ACTION Wait_for_Part_action:
State:=STATE_RUN;
ProcessMessage01:='1IM9';(*warte auf Teil in Stopper*)
Delay.IN:=ST03_571_B69_6.BitInToCheck; 		(*  ISK an stopper.*)
Delay.PT:=T#500ms;
Delay();
END_ACTION

ACTION Wait_for_Part_exit:
ProcessMessage01:='';
END_ACTION

ACTION Close_Seperator_action:
ST03_572_Y70_0.MoveWork:=TRUE;		(* Förderband  Zuführung Vereinzler AST/GST *)
END_ACTION

ACTION Open_Stopper_action:
ST03_572_Y70_1.MoveWork:=TRUE;		(* Förderband  Züführung Stopper AST/GST *)
END_ACTION

ACTION Wait_for_Part__entry:
ProcessMessage01:='';
Delay.IN:=FALSE;
Delay();
END_ACTION

ACTION Wait_for_Part__action:
ProcessMessage01:='1IM10';(*warte auf Teil in Abholposition*)
Delay.IN:=ST03_571_B69_7.BitInToCheck; 		 (* ISK auf Abholposition Robi *)
Delay.PT:=T#500ms;
Delay();
END_ACTION

ACTION Wait_for_Part__exit:
ProcessMessage01:='';
END_ACTION

ACTION Close_Stopper_action:
ST03_572_Y70_1.MoveInit:=TRUE;		(* Förderband  Züführung Stopper AST/GST *)
END_ACTION

ACTION Open_Seperator_action:
ST03_572_Y70_0.MoveInit:=TRUE;		(* Förderband  Zuführung Vereinzler AST/GST *)
END_ACTION

ACTION SeqEnd_action:
SFCTime:=TIME_TO_DINT(TIME()-SFCTimeStart);
State:=STATE_WAIT;
END_ACTION

TRANSITION Abholpos leer:
NOT  ST03_571_B69_7.BitInToCheck		(*  ISK auf Abholposition Robi*)
END_TRANSITION

TRANSITION Part Ready:
Delay.Q AND
NOT ST03_571_B69_7.BitInToCheck	AND		(*  ISK auf Abholposition Robi*)
ST03_571_B69_6.BitInToCheck	AND				(*  ISK anwesend am Stoper*)
Robot01.ActualArea <> 4
END_TRANSITION

TRANSITION StateOk:
ST03_572_Y70_0.State=STATE_OK 	(* Förderband  Zuführung Vereinzler AST/GST *)
END_TRANSITION

TRANSITION State Ok:
ST03_572_Y70_1.State=STATE_OK 	(* Förderband  Züführung Stopper AST/GST *)
END_TRANSITION

TRANSITION Part Ready:
Delay.Q AND
Robot01.ActualArea <> 4
END_TRANSITION

TRANSITION State Ok:
ST03_572_Y70_1.State=STATE_OK 	(* Förderband  Züführung Stopper AST/GST *)
END_TRANSITION

TRANSITION StateOk:
ST03_572_Y70_0.State=STATE_OK 	(* Förderband  Zuführung Vereinzler AST/GST *)
END_TRANSITION
END_PROGRAM

(* POU zLibrary/ept/Service/_CallInit, ST *)
PROGRAM _CallInit


VAR



END_VAR
ST00_Init();
ST02_Init();
ST03_Init();

ST08_Init();
END_PROGRAM

(* POU Stations/ST_00/ST00__Init/ST00_Init, ST *)
PROGRAM ST00_Init


VAR


END_VAR
(* ----------------------------------------------------------------------------------------- *)
(* 																				Sicherungen																				 *)
(* ----------------------------------------------------------------------------------------- *)

(* Init ST00_40_F1 Vorsicherungen Leistung iO (DigIn) *)
ST00_40_F1.sInit.InstName                :='ST00_40_F1';
ST00_40_F1.sInit.Description             :='Sicherungsmodul 24VDC iO';
ST00_40_F1.sInit.BitInName               :='-40_F1';
ST00_40_F1.sInit.HomePosSignal           :=1; (* 0: Signal=Low, 1: Signal=High, 2: always  *)
ST00_40_F1.sInit.MaxTime                 :=2000;
ST00_40_F1.sInit.EnableInEveryMode       :=TRUE;

(* ----------------------------------------------------------------------------------------- *)
(* 																				Sicherheit																							 *)
(* ----------------------------------------------------------------------------------------- *)
(* Init ST03_210_S1 Not-Aus 1 Anlage ausgelöst (DigIn) *)
ST03_210_S1.sInit.InstName               :='ST03_210_S1';
ST03_210_S1.sInit.Description            :='Not-Aus 1 Anlage ausgelöst';
ST03_210_S1.sInit.BitInName              :='-210_S1';
ST03_210_S1.sInit.HomePosSignal          :=0; (* 0: Signal=Low, 1: Signal=High, 2: always  *)
ST03_210_S1.sInit.MaxTime                :=10;
ST03_210_S1.sInit.EnableInEveryMode   	 :=TRUE;

(* Init ST08_210_S2 Not-Aus 2 Anlage ausgelöst (DigIn) *)
ST08_210_S2.sInit.InstName               :='ST08_210_S2';
ST08_210_S2.sInit.Description            :='Not-Aus 2 Anlage ausgelöst';
ST08_210_S2.sInit.BitInName              :='-210_S2';
ST08_210_S2.sInit.HomePosSignal          :=1; (* 0: Signal=Low, 1: Signal=High, 2: always  *)
ST08_210_S2.sInit.MaxTime                :=10;
ST08_210_S2.sInit.EnableInEveryMode   	 :=TRUE;

(* Init ST00_X4_16 Not-Halt 2 Tampondrucker (DigIn) *)
ST00_X4_16.sInit.InstName               :='ST00_X4_16';
ST00_X4_16.sInit.Description            :='Not-Halt 2 Tampondrucker ausgelöst';
ST00_X4_16.sInit.BitInName              :='-X_16';
ST00_X4_16.sInit.HomePosSignal          :=0; (* 0: Signal=Low, 1: Signal=High, 2: always  *)
ST00_X4_16.sInit.MaxTime                :=10;
ST00_X4_16.sInit.EnableInEveryMode   	  :=TRUE;

(* Init ST00_200_A1_A1 Not-Aus iO (DigIn) *)
ST00_200_A1_A1.sInit.InstName            :='ST00_200_A1_A1';
ST00_200_A1_A1.sInit.Description         :='Not-Aus iO';
ST00_200_A1_A1.sInit.BitInName           :='-200_A1:A1';
ST00_200_A1_A1.sInit.HomePosSignal       :=1; (* 0: Signal=Low, 1: Signal=High, 2: always  *)
ST00_200_A1_A1.sInit.MaxTime             :=2000;
ST00_200_A1_A1.sInit.EnableInEveryMode   :=TRUE;

(* Init ST00_220_S1 Schutztüre 1 geöffnet (DigIn) *)
ST00_220_S1.sInit.InstName               :='ST00_220_S1';
ST00_220_S1.sInit.Description            :='Schutztüre 1 geöffnet';
ST00_220_S1.sInit.BitInName              :='-220_S1'; 
ST00_220_S1.sInit.HomePosSignal          :=0; (* 0: Signal=Low, 1: Signal=High, 2: always  *) 
ST00_220_S1.sInit.MaxTime                :=10;
ST00_220_S1.sInit.EnableInEveryMode   	 :=TRUE;

(* Init ST00_220_S2 Schutztüre 2 geöffnet (DigIn) *)
ST00_220_S2.sInit.InstName               :='ST00_220_S2';
ST00_220_S2.sInit.Description            :='Schutztüre 1 geöffnet';
ST00_220_S2.sInit.BitInName              :='-220_S2';
ST00_220_S2.sInit.HomePosSignal          :=0; (* 0: Signal=Low, 1: Signal=High, 2: always  *)
ST00_220_S2.sInit.MaxTime                :=10;
ST00_220_S2.sInit.EnableInEveryMode   	 :=TRUE;

(* Init ST00_223_S2_E1 Schutztüre 1 geschlossen (DigIn) *)
ST00_230_S2_E1.sInit.InstName            :='ST00_230_S2_E1';
ST00_230_S2_E1.sInit.Description         :='Schutztüre 1 geschlossen';
ST00_230_S2_E1.sInit.BitInName           :='-230_S2:E1';
ST00_230_S2_E1.sInit.HomePosSignal       :=2;(* :=1 @@@ *) (* 0: Signal=Low, 1: Signal=High, 2: always  *)
ST00_230_S2_E1.sInit.MaxTime             :=10;
ST00_230_S2_E1.sInit.EnableInEveryMode   	 :=TRUE;

(* Init ST00_240_S1 Schutztüre 9 geschlossen (DigIn) *)
ST00_240_S1.sInit.InstName            :='ST00_240_S1';
ST00_240_S1.sInit.Description         :='Schutztüre 9 geschlossen';
ST00_240_S1.sInit.BitInName           :='-240_S1';
ST00_240_S1.sInit.HomePosSignal       :=2;(* :=1 @@@ *) (* 0: Signal=Low, 1: Signal=High, 2: always  *)
ST00_240_S1.sInit.MaxTime             :=2000;
ST00_240_S1.sInit.EnableInEveryMode   	 :=TRUE;

(* Init ST00_226_S1 Hubtüre 1 Schleuse Einlauf STN 8 geschlossen (DigIn) *)
ST00_226_S1.sInit.InstName               :='ST00_226_S1';
ST00_226_S1.sInit.Description            :='Hubtüre 1 Schleuse Einlauf STN 8 geschlossen';
ST00_226_S1.sInit.BitInName              :='+0-226_S1';
ST00_226_S1.sInit.HomePosSignal          :=2; (* 0: Signal=Low, 1: Signal=High, 2: always  *)
ST00_226_S1.sInit.MaxTime                :=2000;
ST00_226_S1.sInit.EnableInEveryMode   	 :=TRUE;

(* Init ST00_226_S2 Hubtüre 2 Schleuse Einlauf STN 8 geschlossen (DigIn) *)
ST00_226_S2.sInit.InstName               :='ST00_226_S2';
ST00_226_S2.sInit.Description            :='Hubtüre 2 Schleuse Einlauf STN 8 geschlossen';
ST00_226_S2.sInit.BitInName              :='+0-226_S2';
ST00_226_S2.sInit.HomePosSignal          :=2; (* 0: Signal=Low, 1: Signal=High, 2: always  *)
ST00_226_S2.sInit.MaxTime                :=3000;
ST00_226_S2.sInit.EnableInEveryMode   	 :=TRUE;

(* Init ST00_227_S1 Hubtüre 3 Schleuse Auslauf STN 8 geschlossen (DigIn) *) 
ST00_227_S1.sInit.InstName               :='ST00_227_S1';
ST00_227_S1.sInit.Description            :='Hubtüre 3 Schleuse Auslauf STN 8 geschlossen';
ST00_227_S1.sInit.BitInName              :='+0-227_S1';
ST00_227_S1.sInit.HomePosSignal          :=2; (* 0: Signal=Low, 1: Signal=High, 2: always  *)
ST00_227_S1.sInit.MaxTime                :=2000;
ST00_227_S1.sInit.EnableInEveryMode   	 :=TRUE;

(* Init ST00_227_S2 Hubtüre 4 Schleuse Auslauf STN 8 geschlossen (DigIn) *)
ST00_227_S2.sInit.InstName               :='ST00_227_S2';
ST00_227_S2.sInit.Description            :='Hubtüre 4 Schleuse Auslauf STN 8 geschlossen';
ST00_227_S2.sInit.BitInName              :='+0-227_S2';
ST00_227_S2.sInit.HomePosSignal          :=2; (* 0: Signal=Low, 1: Signal=High, 2: always  *)
ST00_227_S2.sInit.MaxTime                :=2000;
ST00_227_S2.sInit.EnableInEveryMode   	 :=TRUE;

(* Init ST00_229_S1 Schutztüre Einlauf Tray STN 8 geschlossen (DigIn) *)
ST00_229_S1.sInit.InstName               :='ST00_229_S1';
ST00_229_S1.sInit.Description            :='Schutztüre Einlauf Tray STN 8 geschlossen';
ST00_229_S1.sInit.BitInName              :='+0-229_S1';
ST00_229_S1.sInit.HomePosSignal          :=2; (* 0: Signal=Low, 1: Signal=High, 2: always  *)
ST00_229_S1.sInit.MaxTime                :=2000;
ST00_229_S1.sInit.EnableInEveryMode   	 :=TRUE;

(* Init ST00_230_S1 Schutztüre Einlauf Tray STN 8 geschlossen (DigIn) *)
ST00_230_S1.sInit.InstName               :='ST00_230_S1';
ST00_230_S1.sInit.Description            :='Schutztüre Auslauf Tray STN 8 geschlossen';
ST00_230_S1.sInit.BitInName              :='+0-230_S1';
ST00_230_S1.sInit.HomePosSignal          :=2; (* 0: Signal=Low, 1: Signal=High, 2: always  *)
ST00_230_S1.sInit.MaxTime                :=2000;
ST00_230_S1.sInit.EnableInEveryMode   	 :=TRUE;

(* Init ST00_231_S1 Schutztüre Panel / Rutsche STN 8 geschlossen (DigIn) *)
ST00_231_S1.sInit.InstName               :='ST00_231_S1';
ST00_231_S1.sInit.Description            :='Schutztüre Panel / Rutsche STN 8 geschlossen';
ST00_231_S1.sInit.BitInName              :='+0-231_S1';
ST00_231_S1.sInit.HomePosSignal          :=2; (* 0: Signal=Low, 1: Signal=High, 2: always  *)
ST00_231_S1.sInit.MaxTime                :=2000;
ST00_231_S1.sInit.EnableInEveryMode   	 :=TRUE;

(* Init ST00_232_S1 Schutztüre 8 Auslauf Trays STN 8 geschlossen (DigIn) *)
ST00_232_S1.sInit.InstName               :='ST00_232_S1';
ST00_232_S1.sInit.Description            :='Schutztüre 8 Auslauf Trays STN 8 geschlossen';
ST00_232_S1.sInit.BitInName              :='+0-232_S1';
ST00_232_S1.sInit.HomePosSignal          :=2; (* 0: Signal=Low, 1: Signal=High, 2: always  *)
ST00_232_S1.sInit.MaxTime                :=2000;
ST00_232_S1.sInit.EnableInEveryMode   	 :=TRUE;

(* Init ST00_170_Motorschutz (DigIn) *)
ST00_170_Motorschutz.sInit.InstName              :='ST00_170_Motorschutz';
ST00_170_Motorschutz.sInit.Description            :='Motorschutz';
ST00_170_Motorschutz.sInit.BitInName              :='+0-170_Motorschutz';
ST00_170_Motorschutz.sInit.HomePosSignal          :=1; (* 0: Signal=Low, 1: Signal=High, 2: always  *)
ST00_170_Motorschutz.sInit.MaxTime                :=2000;
ST00_170_Motorschutz.sInit.EnableInEveryMode   	 :=TRUE;

(* Init ST00_170_Thermokontakt (DigIn) *)
ST00_170_Thermokont.sInit.InstName              :='ST00_170_Thermokont';
ST00_170_Thermokont.sInit.Description            :='Thermokontakt';
ST00_170_Thermokont.sInit.BitInName              :='+0-170_Thermokont';
ST00_170_Thermokont.sInit.HomePosSignal          :=1; (* 0: Signal=Low, 1: Signal=High, 2: always  *)
ST00_170_Thermokont.sInit.MaxTime                :=2000;
ST00_170_Thermokont.sInit.EnableInEveryMode   	 :=TRUE;

(* Init ST00_228_S1 Hubtüre 4 Schleuse Auslauf STN 8 geschlossen (DigIn) *)
ST00_228_S1.sInit.InstName               :='ST00_228_S1';
ST00_228_S1.sInit.Description            :='Pallettierer in Position';
ST00_228_S1.sInit.BitInName              :='+0-228_S1';
ST00_228_S1.sInit.HomePosSignal          :=2; (* 0: Signal=Low, 1: Signal=High, 2: always  *)
ST00_228_S1.sInit.MaxTime                :=2000;
ST00_228_S1.sInit.EnableInEveryMode   	 :=TRUE;


(* Init ST00_71_X1_3 Schnittstelle Bedrucken Tinte JSK auf Übergabeposition (DigIn) *)
ST00_71_X1_3.sInit.InstName            :='ST00_71_X1_3';
ST00_71_X1_3.sInit.Description         :='Bedrucken Tinte JSK auf Übergabeposition';
ST00_71_X1_3.sInit.BitInName           :='-71_X1_3';
ST00_71_X1_3.sInit.HomePosSignal       :=2; (* 0: Signal=Low, 1: Signal=High, 2: always  *)
ST00_71_X1_3.sInit.MaxTime             :=2000;
ST00_71_X1_3.sInit.EnableInEveryMode   :=FALSE;

(* Init ST00_71_X1_4 Schnittstelle Bedrucken Tinte Druckstation betriebsbereit (DigIn) *)
ST00_71_X1_4.sInit.InstName            :='ST00_71_X1_4';
ST00_71_X1_4.sInit.Description         :='Bedrucken Tinte Druckstation betriebsbereit';
ST00_71_X1_4.sInit.BitInName           :='-71_X1_4';
ST00_71_X1_4.sInit.HomePosSignal       :=2; (* 0: Signal=Low, 1: Signal=High, 2: always  *)
ST00_71_X1_4.sInit.MaxTime             :=2000;
ST00_71_X1_4.sInit.EnableInEveryMode   :=FALSE;

(* Init ST00_72_X1_3 Schnittstelle Tampondrucker Teil in Abholposition (DigIn) *)(*Band Entnahmeposition 1*)
ST00_72_X1_3.sInit.InstName            :='ST00_72_X1_3';
ST00_72_X1_3.sInit.Description         :='Band Entnahmeposition 1';
ST00_72_X1_3.sInit.BitInName           :='-72_X1_3';
ST00_72_X1_3.sInit.HomePosSignal       :=2; (* 0: Signal=Low, 1: Signal=High, 2: always  *)
ST00_72_X1_3.sInit.MaxTime             :=2000;
ST00_72_X1_3.sInit.EnableInEveryMode   :=FALSE;

(* Init ST00_72_X1_8 Schnittstelle Tampondrucker Druck abgeschlossen (DigIn) *)
ST00_72_X1_8.sInit.InstName            :='ST00_72_X1_8';
ST00_72_X1_8.sInit.Description         :='Tampondrucker Druck abgeschlossen';
ST00_72_X1_8.sInit.BitInName           :='-72_X1_8';
ST00_72_X1_8.sInit.HomePosSignal       :=2; (* 0: Signal=Low, 1: Signal=High, 2: always  *)
ST00_72_X1_8.sInit.MaxTime             :=2000;
ST00_72_X1_8.sInit.EnableInEveryMode   :=FALSE;

(* Init ST00_292_S1_STOP Bedienstelle Produktion Stop (DigIn) *)
ST00_292_S1_STOP.sInit.InstName          :='ST00_292_S1_STOP';
ST00_292_S1_STOP.sInit.Description       :='Bedienstelle Produktion Stop';
ST00_292_S1_STOP.sInit.BitInName         :='-292_S1:STOP';
ST00_292_S1_STOP.sInit.HomePosSignal     :=2; (* 0: Signal=Low, 1: Signal=High, 2: always  *)
ST00_292_S1_STOP.sInit.MaxTime           :=2000;
ST00_292_S1_STOP.sInit.EnableInEveryMode   	 :=TRUE;

(* Init ST00_292_S2_START Bedienstelle Produktion Start (DigIn) *)
ST00_292_S2_START.sInit.InstName         :='ST00_292_S2_START';
ST00_292_S2_START.sInit.Description      :='Bedienstelle Produktion Start';
ST00_292_S2_START.sInit.BitInName        :='-292_S2:START';
ST00_292_S2_START.sInit.HomePosSignal    :=2; (* 0: Signal=Low, 1: Signal=High, 2: always  *)
ST00_292_S2_START.sInit.MaxTime          :=2000;
ST00_292_S2_START.sInit.EnableInEveryMode   	 :=TRUE;

(* Init ST00_292_S3_RESET Bedienstelle Produktion Start (DigIn) *)
ST00_292_S3_RESET.sInit.InstName         :='ST00_292_S3_RESET';
ST00_292_S3_RESET.sInit.Description      :='Bedienstelle Produktion Reset';
ST00_292_S3_RESET.sInit.BitInName        :='-292_S3:RESET';
ST00_292_S3_RESET.sInit.HomePosSignal    :=2; (* 0: Signal=Low, 1: Signal=High, 2: always  *)
ST00_292_S3_RESET.sInit.MaxTime          :=2000;
ST00_292_S3_RESET.sInit.EnableInEveryMode   	 :=TRUE;

(* Init ST00_350_B20_0 Druckschalter Wartungseinheit Hauptluft min.6 bar (DigIn) *)
ST00_350_B20_0.sInit.InstName            :='ST00_350_B20_0';
ST00_350_B20_0.sInit.Description         :='Druckschalter Wartungseinheit Hauptluft min.6 bar';
ST00_350_B20_0.sInit.BitInName           :='-350_B20.0';
ST00_350_B20_0.sInit.HomePosSignal       :=2; (* 0: Signal=Low, 1: Signal=High, 2: always  *)
ST00_350_B20_0.sInit.MaxTime             :=2000;
ST00_350_B20_0.sInit.EnableInEveryMode   :=TRUE;

(* Init 	ST00_245_V1		Verriegelung Schutztüren-Leuchte (DigOutIn) *)
ST00_245_V1.sInit.InstName           :='ST00_245_V1';
ST00_245_V1.sInit.Description        :='Verriegelung Schutztüren';
ST00_245_V1.sInit.BitOutName         :='-245-V1';
ST00_245_V1.sInit.BitInName          :='';
ST00_245_V1.sInit.HomePosOutput      :=2; (* 0: Signal=Low, 1: Signal=High, 2: always  *)
ST00_245_V1.sInit.MaxTime            :=2000;
ST00_245_V1.sInit.EnableInEveryMode  :=TRUE;

(* Init 	ST00_245_V2_START		Bedienstelle Start-Leuchte (DigOutIn) *)
ST00_245_V2_START.sInit.InstName         :='ST00_245_V2_START';
ST00_245_V2_START.sInit.Description      :='Bedienstelle Start-Leuchte';
ST00_245_V2_START.sInit.BitOutName       :='-245_V2:START';
ST00_245_V2_START.sInit.BitInName        :='';
ST00_245_V2_START.sInit.HomePosOutput    :=2; (* 0: Signal=Low, 1: Signal=High, 2: always  *)
ST00_245_V2_START.sInit.MaxTime          :=2000;
ST00_245_V2_START.sInit.EnableInEveryMode   	 :=TRUE;

(* Init 	ST00_245_V3_RESET		Bedienstelle Reset-Schutztüren-Leuchte (DigOutIn) *)
ST00_245_V3_RESET.sInit.InstName         :='ST00_245_V3_RESET';
ST00_245_V3_RESET.sInit.Description      :='Bedienstelle Reset-Leuchte';
ST00_245_V3_RESET.sInit.BitOutName       :='-245_V3:RESET';
ST00_245_V3_RESET.sInit.BitInName        :='';
ST00_245_V3_RESET.sInit.HomePosOutput    :=2; (* 0: Signal=Low, 1: Signal=High, 2: always  *)
ST00_245_V3_RESET.sInit.MaxTime          :=2000;
ST00_245_V3_RESET.sInit.EnableInEveryMode:=TRUE;

(* Init 	ST00_245_S1_STOP 	Bedienstelle Produktion Stop (DigIn) *)
ST00_245_S1_STOP.sInit.InstName          :='ST00_245_S1_STOP';
ST00_245_S1_STOP.sInit.Description       :='Bedienstelle Produktion Stop';
ST00_245_S1_STOP.sInit.BitInName         :='-245_S1:STOP';
ST00_245_S1_STOP.sInit.HomePosSignal     :=2; (* 0: Signal=Low, 1: Signal=High, 2: always  *)
ST00_245_S1_STOP.sInit.MaxTime           :=2000;
ST00_245_S1_STOP.sInit.EnableInEveryMode :=TRUE;

(* Init 	ST00_245_S2_START	Bedienstelle Produktion Start (DigIn) *)
ST00_245_S2_START.sInit.InstName         :='ST00_245_S2_START';
ST00_245_S2_START.sInit.Description      :='Bedienstelle Produktion Start';
ST00_245_S2_START.sInit.BitInName        :='-245_S2:START';
ST00_245_S2_START.sInit.HomePosSignal    :=2; (* 0: Signal=Low, 1: Signal=High, 2: always  *)
ST00_245_S2_START.sInit.MaxTime          :=2000;
ST00_245_S2_START.sInit.EnableInEveryMode:=TRUE;

(* Init 	ST00_245_S3_RESET	Bedienstelle Produktion Reset (DigIn) *)
ST00_245_S3_RESET.sInit.InstName         :='ST00_245_S3_RESET';
ST00_245_S3_RESET.sInit.Description      :='Bedienstelle Produktion Reset';
ST00_245_S3_RESET.sInit.BitInName        :='-245_S3:RESET';
ST00_245_S3_RESET.sInit.HomePosSignal    :=2; (* 0: Signal=Low, 1: Signal=High, 2: always  *)
ST00_245_S3_RESET.sInit.MaxTime			 :=2000;
ST00_245_S3_RESET.sInit.EnableInEveryMode:=TRUE;


(* ----------------------------------------------------------------------------------------- *)
(* 																			Ausgänge																						 *)
(* ----------------------------------------------------------------------------------------- *)

(* Init ST00_31_K1 Beleuchtung Anlage (DigOutIn) *)
ST00_31_K1.sInit.InstName                :='ST00_31_K1';
ST00_31_K1.sInit.Description             :='Beleuchtung Anlage';
ST00_31_K1.sInit.BitOutName              :='-31_K1'; 
ST00_31_K1.sInit.BitInName               :='';
ST00_31_K1.sInit.HomePosOutput           :=2; (* 0: Signal=Low, 1: Signal=High, 2: always  *)
ST00_31_K1.sInit.MaxTime                 :=2000;
ST00_31_K1.sInit.EnableInEveryMode   	 	:=TRUE;
ST00_31_K1.sInit.EnableVisuInEveryMode   :=TRUE;

(* Init ST00_350_H1 Signalsäule RD Maschine Alarm/Störung (DigOutIn) *)
ST00_350_H1.sInit.InstName               :='ST00_350_H1';
ST00_350_H1.sInit.Description            :='Signalsäule RD Maschine Alarm/Störung';
ST00_350_H1.sInit.BitOutName             :='-350_H1'; 
ST00_350_H1.sInit.BitInName              :=''; 
ST00_350_H1.sInit.HomePosOutput          :=2; (* 0: Signal=Low, 1: Signal=High, 2: always  *)
ST00_350_H1.sInit.MaxTime                :=2000;
ST00_350_H1.sInit.EnableInEveryMode   	 :=TRUE;

(* Init ST00_350_H2 Signalsäule YE Bedienereingriff erforderlich (DigOutIn) *)
ST00_350_H2.sInit.InstName               :='ST00_350_H2';
ST00_350_H2.sInit.Description            :='Signalsäule YE Bedienereingriff erforderlich';
ST00_350_H2.sInit.BitOutName             :='-350_H2';
ST00_350_H2.sInit.BitInName              :='';
ST00_350_H2.sInit.HomePosOutput          :=2; (* 0: Signal=Low, 1: Signal=High, 2: always  *)
ST00_350_H2.sInit.MaxTime                :=2000;
ST00_350_H2.sInit.EnableInEveryMode   	 :=TRUE;

(* Init ST00_350_H3 Signalsäule GN Maschine Automatik (DigOutIn) *)
ST00_350_H3.sInit.InstName               :='ST00_350_H3';
ST00_350_H3.sInit.Description            :='Signalsäule GN Maschine Automatik';
ST00_350_H3.sInit.BitOutName             :='-350_H3'; 
ST00_350_H3.sInit.BitInName              :=''; 
ST00_350_H3.sInit.HomePosOutput          :=2; (* 0: Signal=Low, 1: Signal=High, 2: always  *)
ST00_350_H3.sInit.MaxTime                :=2000;
ST00_350_H3.sInit.EnableInEveryMode   	 :=TRUE;

(* Init ST00_200_A1_E4 Quittierung Not-Aus (DigOutIn) *)
ST00_200_A1_E4.sInit.InstName            :='ST00_200_A1_E4';
ST00_200_A1_E4.sInit.Description         :='Quittierung Not-Aus';
ST00_200_A1_E4.sInit.BitOutName          :='-200_A1:E4'; 
ST00_200_A1_E4.sInit.BitInName           :=''; 
ST00_200_A1_E4.sInit.HomePosSignal       :=0; (* 0: Signal=Low, 1: Signal=High, 2: always  *)
ST00_200_A1_E4.sInit.MaxTime             :=2000;
ST00_200_A1_E4.sInit.EnableInEveryMode   :=TRUE;
ST00_200_A1_E4.sInit.EnableVisuInEveryMode :=TRUE;

(* Init ST00_220_S1_S31 Verriegelung Schutztüren (DigOutIn) *)
ST00_220_S1_S31.sInit.InstName           :='ST00_220_S1_S31';
ST00_220_S1_S31.sInit.Description        :='Verriegelung Schutztüren';
ST00_220_S1_S31.sInit.BitOutName         :='-220-S1:S31';
ST00_220_S1_S31.sInit.BitInName          :='';
ST00_220_S1_S31.sInit.HomePosOutput      :=2; (* 0: Signal=Low, 1: Signal=High, 2: always  *)
ST00_220_S1_S31.sInit.MaxTime            :=2000;
ST00_220_S1_S31.sInit.EnableInEveryMode   	 :=TRUE;

(* Init ST00_292_H2_START Bedienstelle Start-Leuchte (DigOutIn) *)
ST00_292_H2_START.sInit.InstName         :='ST00_292_H2_START';
ST00_292_H2_START.sInit.Description      :='Bedienstelle Start-Leuchte';
ST00_292_H2_START.sInit.BitOutName       :='-292_H2:START';
ST00_292_H2_START.sInit.BitInName        :='';
ST00_292_H2_START.sInit.HomePosOutput    :=2; (* 0: Signal=Low, 1: Signal=High, 2: always  *)
ST00_292_H2_START.sInit.MaxTime          :=2000;
ST00_292_H2_START.sInit.EnableInEveryMode   	 :=TRUE;

(* Init ST00_292_H3_RESET Bedienstelle Reset-Leuchte (DigOutIn) *)
ST00_292_H3_RESET.sInit.InstName         :='ST00_292_H3_RESET';
ST00_292_H3_RESET.sInit.Description      :='Bedienstelle Reset-Leuchte';
ST00_292_H3_RESET.sInit.BitOutName       :='-292_H3:RESET';
ST00_292_H3_RESET.sInit.BitInName        :='';
ST00_292_H3_RESET.sInit.HomePosOutput    :=2; (* 0: Signal=Low, 1: Signal=High, 2: always  *)
ST00_292_H3_RESET.sInit.MaxTime          :=2000;
ST00_292_H3_RESET.sInit.EnableInEveryMode   	 :=TRUE;

(* Init ST00_71_K2 Schnittstelle Bedrucken Tinte Abholposition frei (DigOutIn) *)
ST00_71_K2.sInit.InstName             :='ST00_71_K2';
ST00_71_K2.sInit.Description          :='Bedrucken Tinte Abholposition frei';
ST00_71_K2.sInit.BitOutName           :='-71_K1';
ST00_71_K2.sInit.BitInName            :='';
ST00_71_K2.sInit.HomePosSignal        :=2; (* 0: Signal=Low, 1: Signal=High, 2: always  *)
ST00_71_K2.sInit.HomePosOutput	 :=2; (* 0: Signal=Low, 1: Signal=High, 2: always  *)
ST00_71_K2.sInit.MaxTime              :=2000;
ST00_71_K2.sInit.EnableVisuInEveryMode:=TRUE;

(* Schnittstelle Förderband frei für Spritzmaschine(DigOutIn) *)
ST00_73_K3.sInit.InstName             :='ST00_73_K3';
ST00_73_K3.sInit.Description          :='Förderband frei für Spritzmaschine';
ST00_73_K3.sInit.BitOutName           :='-73_K3';
ST00_73_K3.sInit.BitInName            :='';
ST00_73_K3.sInit.HomePosSignal        :=2; (* 0: Signal=Low, 1: Signal=High, 2: always  *)
ST00_73_K3.sInit.HomePosOutput				:=2; (* 0: Signal=Low, 1: Signal=High, 2: always  *)
ST00_73_K3.sInit.MaxTime              :=2000;

(*ST00_73_K4  Schnittstelle Freigabe von Spritzmaschine (nur für Anlagen ohne Rundtisch) (DigIn)*)
ST00_73_K4.sInit.InstName                :='ST00_73_K4';
ST00_73_K4.sInit.Description             :=' Freigabe Spritzmaschine';
ST00_73_K4.sInit.BitInName               :='-73_K4';
ST00_73_K4.sInit.HomePosSignal   	 :=2; (* 0: Signal=Low, 1: Signal=High, 2: always  *)
ST00_73_K4.sInit.MaxTime                 :=2000;

(* Init ST00_74_B7_2 Stopper GST1 DS (ValveSensor) *)
ST00_74_B7_2.sInit.InstName            :='ST00_74_B7_2';
ST00_74_B7_2.sInit.BitName            :='+0_74_B7_2';
ST00_74_B7_2.sInit.Description         :='Stopper GST1 DS';
ST00_74_B7_2.sInit.SensorType          :=sValveSensorType_INIT;

(* Init ST00_74_B7_3 Stopper GST1 DS (ValveSensor) *)
ST00_74_B7_3.sInit.InstName            :='ST00_74_B7_3';
ST00_74_B7_3.sInit.BitName            :='+0_74_B7_3';
ST00_74_B7_3.sInit.Description         :='Stopper GST2 PS';
ST00_74_B7_3.sInit.SensorType          :=sValveSensorType_INIT;

(* Init ST00_74_B7_4 Vereinzeler AST1 DS (ValveSensor) *)
ST00_74_B7_4.sInit.InstName            :='ST00_74_B7_4';
ST00_74_B7_4.sInit.BitName            :='+0_74_B7_4';
ST00_74_B7_4.sInit.Description         :='Vereinzeler GST1 DS';
ST00_74_B7_4.sInit.SensorType          :=sValveSensorType_INIT;

(* Init ST00_74_B7_5 Vereinzeler AST2 PS (ValveSensor) *)
ST00_74_B7_5.sInit.InstName            :='ST00_74_B7_5';
ST00_74_B7_5.sInit.BitName            :='+0_74_B7_5';
ST00_74_B7_5.sInit.Description         :='Vereinzeler GST2 PS';
ST00_74_B7_5.sInit.SensorType          :=sValveSensorType_INIT;

(* Init ST00_74_B7_6  Vereinzeler GST1 DS(ValveSensor) *)
ST00_74_B7_6.sInit.InstName            :='ST00_74_B7_6';
ST00_74_B7_6.sInit.BitName            :='+0_74_B7_6';
ST00_74_B7_6.sInit.Description         :='Vereinzeler AST1 DS';
ST00_74_B7_6.sInit.SensorType          :=sValveSensorType_WORK;

(* Init ST00_74_B7_7 Vereinzeler GST2 PS (ValveSensor) *)
ST00_74_B7_7.sInit.InstName            :='ST00_74_B7_7';
ST00_74_B7_7.sInit.BitName            :='+0_74_B7_7';
ST00_74_B7_7.sInit.Description         :='Vereinzeler AST2 PS';
ST00_74_B7_7.sInit.SensorType          :=sValveSensorType_WORK;

(* Init ST00_74_Y2_4 Stopper ISK (lt. Schaltplan 62Y1)(Valve) *)
ST00_74_Y2_4.sInit.InstName            :='ST00_74_Y2_4';
ST00_74_Y2_4.sInit.BitName            :='+0_74_Y2_4';
ST00_74_Y2_4.sInit.Description         :='Stopper Bandstrecke';
ST00_74_Y2_4.sInit.HomePosDefine       :=HOME_ALWAYS;
ST00_74_Y2_4.sInit.InitDescription     :='GS';
ST00_74_Y2_4.sInit.WorkDescription     :='AS';
ST00_74_Y2_4.sInit.DampBothTime        :=200;
ST00_74_Y2_4.sInit.KindOfValve         :='A';
ST00_74_Y2_4.sInit.MaxTime             :=2000;

(* Init ST00_74_Y2_5 Vereinzeler ISK (lt. Schaltplan 62Y3)(Valve) *)
ST00_74_Y2_5.sInit.InstName            :='ST00_74_Y2_5';
ST00_74_Y2_5.sInit.BitName            :='+0_74_Y2_5';
ST00_74_Y2_5.sInit.Description         :='Vereinzeler Bandstrecke';
ST00_74_Y2_5.sInit.HomePosDefine       :=HOME_ALWAYS;
ST00_74_Y2_5.sInit.InitDescription     :='GS';
ST00_74_Y2_5.sInit.WorkDescription     :='AS';
ST00_74_Y2_5.sInit.DampBothTime        :=200;
ST00_74_Y2_5.sInit.KindOfValve         :='A';
ST00_74_Y2_5.sInit.MaxTime             :=2000;
END_PROGRAM

(* POU Stations/ST_02_RT_Tampondrucker/ST02__Init/ST02_Init, ST *)
PROGRAM ST02_Init


VAR


END_VAR
(* ----------------------------------------------------------------------------------------- *)

(* Init ST02_S1_6A01 ST02 Sicherung 24V  (DigIn) *)
ST02_S1_6A01.sInit.InstName                :='ST02_S1_6A01';
ST02_S1_6A01.sInit.Description             :='Sicherungsmodul 24VDC';
ST02_S1_6A01.sInit.BitInName               :='-S1_6A01';
ST02_S1_6A01.sInit.HomePosSignal   :=1; (* 0: Signal=Low, 1: Signal=High, 2: always  *)
ST02_S1_6A01.sInit.MaxTime                 :=2000;
ST02_S1_6A01.sInit.EnableInEveryMode       :=TRUE;

(* ----------------------------------------------------------------------------------------- *)
(* ----------------------------------------------------------------------------------------- *)
(* Init ST02_FDB_55X1_5_READY IFM Kamera Flügelerkennung links Ready (DigIn) *)
ST02_FDB_55X1_5_READY.sInit.InstName          :='ST02_FDB_55X1_5_READY';
ST02_FDB_55X1_5_READY.sInit.Description       :='IFM Kamera links ready';
ST02_FDB_55X1_5_READY.sInit.BitInName         :='+55X1_5_READY';
ST02_FDB_55X1_5_READY.sInit.HomePosSignal     :=2; (* 0: Signal=Low, 1: Signal=High, 2: always  *)
ST02_FDB_55X1_5_READY.sInit.MaxTime           :=2000;

(* Init ST02_FDB_55X1_6_IO IFM Kamera Flügelerkennung links Ergebnis iO (DigIn) *)
ST02_FDB_55X1_6_IO.sInit.InstName          :='ST02_FDB_55X1_6_IO';
ST02_FDB_55X1_6_IO.sInit.Description       :='IFM Kamera links Ergebnis iO';
ST02_FDB_55X1_6_IO.sInit.BitInName         :='+55X1_6_IO';
ST02_FDB_55X1_6_IO.sInit.HomePosSignal     :=2; (* 0: Signal=Low, 1: Signal=High, 2: always  *)
ST02_FDB_55X1_6_IO.sInit.MaxTime           :=2000;

(* Init ST02_FDB_55X1_6_NIO IFM Kamera Flügelerkennung links Ergebnis niO (DigIn) *)
ST02_FDB_55X1_6_NIO.sInit.InstName          :='ST02_FDB_55X1_6_NIO';
ST02_FDB_55X1_6_NIO.sInit.Description       :='IFM Kamera links Ergebnis niO';
ST02_FDB_55X1_6_NIO.sInit.BitInName         :='+55X1_6_NIO';
ST02_FDB_55X1_6_NIO.sInit.HomePosSignal     :=2; (* 0: Signal=Low, 1: Signal=High, 2: always  *)
ST02_FDB_55X1_6_NIO.sInit.MaxTime           :=2000;

(* Init ST02_FDB_55X1_2_TRIGGER IFM Kamera Flügelerkennung links Trigger (DigOutIn) *)
ST02_FDB_55X1_2_TRIGGER.sInit.InstName          :='ST02_FDB_55X1_2_TRIGGER';
ST02_FDB_55X1_2_TRIGGER.sInit.Description       :='IFM Kamera links Trigger';
ST02_FDB_55X1_2_TRIGGER.sInit.BitOutName        :='+55X1_2_TRIGGER';
ST02_FDB_55X1_2_TRIGGER.sInit.BitInName         :='';
ST02_FDB_55X1_2_TRIGGER.sInit.HomePosSignal     :=2; (* 0: Signal=Low, 1: Signal=High, 2: always  *)
ST02_FDB_55X1_2_TRIGGER.sInit.MaxTime           :=2000;

(* Init ST02_FDB_55X1_7_JOB_BIT1 IFM Kamera links Jobwechsel Bit1 (DigOutIn) *)
ST02_FDB_55X1_7_JOB_BIT1.sInit.InstName          :='ST02_FDB_55X1_7_JOB_BIT1';
ST02_FDB_55X1_7_JOB_BIT1.sInit.Description       :='IFM Kamera  Job Bit 1';
ST02_FDB_55X1_7_JOB_BIT1.sInit.BitOutName        :='+55X1_7_JOB_BIT1';
ST02_FDB_55X1_7_JOB_BIT1.sInit.BitInName         :='';
ST02_FDB_55X1_7_JOB_BIT1.sInit.HomePosSignal     :=2; (* 0: Signal=Low, 1: Signal=High, 2: always  *)
ST02_FDB_55X1_7_JOB_BIT1.sInit.MaxTime           :=2000;

(* Init ST02_FDB_55X1_7_JOB_BIT2 IFM Kamera links Jobwechsel Bit2 (DigOutIn) *)
ST02_FDB_55X1_7_JOB_BIT2.sInit.InstName          :='ST02_FDB_55X1_7_JOB_BIT2';
ST02_FDB_55X1_7_JOB_BIT2.sInit.Description       :='IFM Kamera  Job Bit 2';
ST02_FDB_55X1_7_JOB_BIT2.sInit.BitOutName        :='+55X1_7_JOB_BIT2';
ST02_FDB_55X1_7_JOB_BIT2.sInit.BitInName         :='';
ST02_FDB_55X1_7_JOB_BIT2.sInit.HomePosSignal     :=2; (* 0: Signal=Low, 1: Signal=High, 2: always  *)
ST02_FDB_55X1_7_JOB_BIT2.sInit.MaxTime           :=2000;
(* Init ST02_FDB_56X1_5_READY IFM Kamera Flügelerkennung rechts Ready (DigIn) *)
ST02_FDB_56X1_5_READY.sInit.InstName          :='ST02_FDB_56X1_5_READY';
ST02_FDB_56X1_5_READY.sInit.Description       :='IFM Kamera rechts ready';
ST02_FDB_56X1_5_READY.sInit.BitInName         :='+56X1_5_READY';
ST02_FDB_56X1_5_READY.sInit.HomePosSignal     :=2; (* 0: Signal=Low, 1: Signal=High, 2: always  *)
ST02_FDB_56X1_5_READY.sInit.MaxTime           :=2000;

(* Init ST02_FDB_56X1_6_IO IFM Kamera Flügelerkennung rechts Ergebnis iO (DigIn) *)
ST02_FDB_56X1_6_IO.sInit.InstName          :='ST02_FDB_56X1_6_IO';
ST02_FDB_56X1_6_IO.sInit.Description       :='IFM Kamera rechts Ergebnis iO';
ST02_FDB_56X1_6_IO.sInit.BitInName         :='+56X1_6_IO';
ST02_FDB_56X1_6_IO.sInit.HomePosSignal     :=2; (* 0: Signal=Low, 1: Signal=High, 2: always  *)
ST02_FDB_56X1_6_IO.sInit.MaxTime           :=2000;

(* Init ST02_FDB_56X1_6_NIO IFM Kamera Flügelerkennung rechts Ergebnis niO (DigIn) *)
ST02_FDB_56X1_6_NIO.sInit.InstName          :='ST02_FDB_56X1_6_NIO';
ST02_FDB_56X1_6_NIO.sInit.Description       :='IFM Kamera rechts Ergebnis niO';
ST02_FDB_56X1_6_NIO.sInit.BitInName         :='+56X1_6_NIO';
ST02_FDB_56X1_6_NIO.sInit.HomePosSignal     :=2; (* 0: Signal=Low, 1: Signal=High, 2: always  *)
ST02_FDB_56X1_6_NIO.sInit.MaxTime           :=2000;

(* Init ST02_FDB_56X1_2_TRIGGER IFM Kamera Flügelerkennung rechts Trigger (DigOutIn) *)
ST02_FDB_56X1_2_TRIGGER.sInit.InstName          :='ST02_FDB_56X1_2_TRIGGER';
ST02_FDB_56X1_2_TRIGGER.sInit.Description       :='IFM Kamera rechts Trigger';
ST02_FDB_56X1_2_TRIGGER.sInit.BitOutName        :='+56X1_2_TRIGGER';
ST02_FDB_56X1_2_TRIGGER.sInit.BitInName         :='';
ST02_FDB_56X1_2_TRIGGER.sInit.HomePosSignal     :=2; (* 0: Signal=Low, 1: Signal=High, 2: always  *)
ST02_FDB_56X1_2_TRIGGER.sInit.MaxTime           :=2000;

(* Init ST02_FDB_56X1_7_JOB_BIT1 IFM Kamera rechts Jobwechsel Bit1 (DigOutIn) *)
ST02_FDB_56X1_7_JOB_BIT1.sInit.InstName          :='ST02_FDB_56X1_7_JOB_BIT1';
ST02_FDB_56X1_7_JOB_BIT1.sInit.Description       :='IFM Kamera  Job Bit 1';
ST02_FDB_56X1_7_JOB_BIT1.sInit.BitOutName        :='+56X1_7_JOB_BIT1';
ST02_FDB_56X1_7_JOB_BIT1.sInit.BitInName         :='';
ST02_FDB_56X1_7_JOB_BIT1.sInit.HomePosSignal     :=2; (* 0: Signal=Low, 1: Signal=High, 2: always  *)
ST02_FDB_56X1_7_JOB_BIT1.sInit.MaxTime           :=2000;

(* Init ST02_FDB_56X1_7_JOB_BIT2 IFM Kamera rechts Jobwechsel Bit2 (DigOutIn) *)
ST02_FDB_56X1_7_JOB_BIT2.sInit.InstName          :='ST02_FDB_56X1_7_JOB_BIT2';
ST02_FDB_56X1_7_JOB_BIT2.sInit.Description       :='IFM Kamera  Job Bit 2';
ST02_FDB_56X1_7_JOB_BIT2.sInit.BitOutName        :='+56X1_7_JOB_BIT2';
ST02_FDB_56X1_7_JOB_BIT2.sInit.BitInName         :='';
ST02_FDB_56X1_7_JOB_BIT2.sInit.HomePosSignal     :=2; (* 0: Signal=Low, 1: Signal=High, 2: always  *)
ST02_FDB_56X1_7_JOB_BIT2.sInit.MaxTime           :=2000;

(* Init ST02_FDB_54_B41 Kamera ISK anwesend an Prüfposition (DigIn) *)
ST02_FDB_54_B41.sInit.InstName          :='ST02_FDB_54_B41';
ST02_FDB_54_B41.sInit.Description       :='Kamera ISK an Prüfposition';
ST02_FDB_54_B41.sInit.BitInName         :='+54B41';
ST02_FDB_54_B41.sInit.HomePosSignal     :=2; (* 0: Signal=Low, 1: Signal=High, 2: always  *)
ST02_FDB_54_B41.sInit.MaxTime           :=2000;

(* Init ST02_DT_65B11 Tampondrucker Nest 1 leer (DigIn) *)
ST02_DT_65B11.sInit.InstName            :='ST02_DT_65B11';
ST02_DT_65B11.sInit.Description         :='Tampondrucker Nest 1 leer';
ST02_DT_65B11.sInit.BitInName           :='+65B11';
ST02_DT_65B11.sInit.HomePosSignal       :=2; (* 0: Signal=Low, 1: Signal=High, 2: always  *)
ST02_DT_65B11.sInit.MaxTime             :=2000;
ST02_DT_65B11.sInit.EnableInEveryMode   :=FALSE;

(* Init ST02_DT_65B21 Tampondrucker Nest 2 leer (DigIn) *)
ST02_DT_65B21.sInit.InstName            :='ST02_DT_65B21';
ST02_DT_65B21.sInit.Description         :='Tampondrucker Nest 2 leer';
ST02_DT_65B21.sInit.BitInName           :='+65B21';
ST02_DT_65B21.sInit.HomePosSignal       :=2; (* 0: Signal=Low, 1: Signal=High, 2: always  *)
ST02_DT_65B21.sInit.MaxTime             :=2000;
ST02_DT_65B21.sInit.EnableInEveryMode   :=FALSE;

(* Init ST02_S1_70K61_A1 Start Bedruckung (DigOutIn) *)
ST02_S1_70K61_A1.sInit.InstName          :='ST02_S1_70K61_A1';
ST02_S1_70K61_A1.sInit.Description       :='Start Bedruckung';
ST02_S1_70K61_A1.sInit.BitOutName        :='+70K61_A1';
ST02_S1_70K61_A1.sInit.BitInName         :='';
ST02_S1_70K61_A1.sInit.HomePosSignal     :=0; (* 0: Signal=Low, 1: Signal=High, 2: always  *)
ST02_S1_70K61_A1.sInit.MaxTime         		:=2000;

(*ST02_S1_40K01 Freigabe Förderband von SPM (DigIn)*)
ST02_S1_40K01.sInit.InstName                :='ST02_S1_40K01';
ST02_S1_40K01.sInit.Description             :=' Freigabe Förderband von SPM';
ST02_S1_40K01.sInit.BitInName               :='-S1_40K01_14';
ST02_S1_40K01.sInit.HomePosSignal    :=2; (* 0: Signal=Low, 1: Signal=High, 2: always  *)
ST02_S1_40K01.sInit.MaxTime                 :=2000;

(* Init ST02_FDB_80_B02 Band Entnahmeposition 2  (DigIn) *)
ST02_FDB_80_B02.sInit.InstName                :='ST02_FDB_80_B02';
ST02_FDB_80_B02.sInit.Description             :=' Band Entnahmeposition 2';
ST02_FDB_80_B02.sInit.BitInName               :='-80_B02';
ST02_FDB_80_B02.sInit.HomePosSignal    :=2; (* 0: Signal=Low, 1: Signal=High, 2: always  *)
ST02_FDB_80_B02.sInit.MaxTime                 :=2000;

(* Init ST02_35_S31 ST02 Druckschalter Wartungseinheit Hauptluft min.6 bar (DigIn) *)
ST02_35_S31.sInit.InstName            :='ST02_35_S31';
ST02_35_S31.sInit.Description         :='ST02 Druckschalter Wartungseinheit Hauptluft min.6 bar';
ST02_35_S31.sInit.BitInName           :='-35_S31';
ST02_35_S31.sInit.HomePosSignal       :=2; (* 0: Signal=Low, 1: Signal=High, 2: always  *)
ST02_35_S31.sInit.MaxTime             :=2000;
ST02_35_S31.sInit.EnableInEveryMode   :=TRUE;

(*---------------------------------------------------------------------------------------------------------------*)
(* Init ST02_62_Y6 Tisch drehen 0 - 180 Grad(Valve) *)
ST02_62_Y6.sInit.InstName            :='ST02_62_Y6';
ST02_62_Y6.sInit.BitName            :='+62Y6';
ST02_62_Y6.sInit.Description         :='Tisch drehen ';
ST02_62_Y6.sInit.HomePosDefine       :=HOME_ALWAYS;
ST02_62_Y6.sInit.InitDescription     :='0 Grad';
ST02_62_Y6.sInit.WorkDescription     :='180 Grad';
ST02_62_Y6.sInit.DampBothTime        :=200;
ST02_62_Y6.sInit.KindOfValve         :='2G';
ST02_62_Y6.sInit.MaxTime             :=2000;

(* Init ST02_FDB_40_B61 Iso von SPM auf Band abgelegt (DigIn) *)
ST02_FDB_40_B61.sInit.InstName            :='ST02_FDB_40_B61';
ST02_FDB_40_B61.sInit.Description         :=' Iso von SPM auf Band abgelegt';
ST02_FDB_40_B61.sInit.BitInName           :='+40B61';
ST02_FDB_40_B61.sInit.HomePosSignal       :=2; (* 0: Signal=Low, 1: Signal=High, 2: always  *)
ST02_FDB_40_B61.sInit.MaxTime             :=2000;
(*ST02_FDB_40_B61.sInit.EnableInEveryMode   :=FALSE;*)

(* Init ST02_FDB_40_B71 Iso auf Band vor Vereinzler (DigIn) *)
ST02_FDB_40_B71.sInit.InstName            :='ST02_FDB_40_B71';
ST02_FDB_40_B71.sInit.Description         :=' Iso auf Band vor Vereinzler';
ST02_FDB_40_B71.sInit.BitInName           :='+40B71';
ST02_FDB_40_B71.sInit.HomePosSignal       :=2; (* 0: Signal=Low, 1: Signal=High, 2: always  *)
ST02_FDB_40_B71.sInit.MaxTime             :=2000;
(*ST02_FDB_40_B71.sInit.EnableInEveryMode   :=FALSE;*)

(* Init ST02_DT_62_B81 Tisch drehen 0 Grad (ValveSensor) *)
ST02_DT_62_B81.sInit.InstName            :='ST02_DT_62_B81';
ST02_DT_62_B81.sInit.BitName            :='+62B81';
ST02_DT_62_B81.sInit.Description         :='Tisch drehen 0 Grad';
ST02_DT_62_B81.sInit.SensorType          :=sValveSensorType_INIT;

(* Init ST02_DT_62_B91 Tisch drehen 180 Grad (ValveSensor) *)
ST02_DT_62_B91.sInit.InstName            :='ST02_DT_62_B91';
ST02_DT_62_B91.sInit.BitName            :='+62B91';
ST02_DT_62_B91.sInit.Description         :='Tisch drehen 180 Grad';
ST02_DT_62_B91.sInit.SensorType          :=sValveSensorType_WORK;

(*---------------------------------------------------------------------------------------------------------------*)
(* Init ST02_62_Y9 Schwenkarm 2 drehen 90 - 180 Grad(Valve) *)
ST02_62_Y9.sInit.InstName            :='ST02_62_Y9';
ST02_62_Y9.sInit.BitName            :='+62Y9';
ST02_62_Y9.sInit.Description         :='Schwenkarm 2 drehen 90 - 180 Grad ';
ST02_62_Y9.sInit.HomePosDefine       :=HOME_ALWAYS;
ST02_62_Y9.sInit.InitDescription     :='90 Grad';
ST02_62_Y9.sInit.WorkDescription     :='180 Grad';
ST02_62_Y9.sInit.DampBothTime        :=200;
ST02_62_Y9.sInit.KindOfValve         :='2G';
ST02_62_Y9.sInit.MaxTime             :=2000;

(* Init ST02_62_Y11 Schwenkarm 2 drehen 90 - 0 Grad(Valve) *)
ST02_62_Y11.sInit.InstName            :='ST02_62_Y11';
ST02_62_Y11.sInit.BitName            :='+62Y11';
ST02_62_Y11.sInit.Description         :='Schwenkarm 2 drehen 90 - 0 Grad ';
ST02_62_Y11.sInit.HomePosDefine       :=HOME_ALWAYS;
ST02_62_Y11.sInit.InitDescription     :='90 Grad';
ST02_62_Y11.sInit.WorkDescription     :='0 Grad';
ST02_62_Y11.sInit.DampBothTime        :=200;
ST02_62_Y11.sInit.KindOfValve         :='2G';
ST02_62_Y11.sInit.MaxTime             :=2000;

(* Init ST02_DT_61_B31 Schwenkarm 2 0 Grad (ValveSensor) *)
ST02_DT_61_B31.sInit.InstName            :='ST02_DT_61_B31';
ST02_DT_61_B31.sInit.BitName            :='+61B31';
ST02_DT_61_B31.sInit.Description         :='Schwenkarm 2 0 Grad';
ST02_DT_61_B31.sInit.SensorType          :=sValveSensorType_WORK;

(* Init ST02_DT_61_B11 Schwenkarm 2 180 Grad (ValveSensor) *)
ST02_DT_61_B11.sInit.InstName            :='ST02_DT_61_B11';
ST02_DT_61_B11.sInit.BitName            :='+61B11';
ST02_DT_61_B11.sInit.Description         :='Schwenkarm 2 180 Grad';
ST02_DT_61_B11.sInit.SensorType          :=sValveSensorType_WORK;

(*---------------------------------------------------------------------------------------------------------------*)
(* Init ST02_62_Y13 Schwenkarm 1 drehen 90 - 180 Grad(Valve) *)
ST02_62_Y13.sInit.InstName            :='ST02_62_Y13';
ST02_62_Y13.sInit.BitName            :='+62Y13';
ST02_62_Y13.sInit.Description         :='Schwenkarm 1 drehen 90 - 180 Grad ';
ST02_62_Y13.sInit.HomePosDefine       :=HOME_ALWAYS;
ST02_62_Y13.sInit.InitDescription     :='90 Grad';
ST02_62_Y13.sInit.WorkDescription     :='180 Grad';
ST02_62_Y13.sInit.DampBothTime        :=200;
ST02_62_Y13.sInit.KindOfValve         :='2G';
ST02_62_Y13.sInit.MaxTime             :=2000;

(* Init ST02_62_Y15 Schwenkarm 1 drehen 90 - 0 Grad(Valve) *)
ST02_62_Y15.sInit.InstName            :='ST02_62_Y15';
ST02_62_Y15.sInit.BitName            :='+62Y15';
ST02_62_Y15.sInit.Description         :='Schwenkarm 1 drehen 90 - 0 Grad ';
ST02_62_Y15.sInit.HomePosDefine       :=HOME_ALWAYS;
ST02_62_Y15.sInit.InitDescription     :='90 Grad';
ST02_62_Y15.sInit.WorkDescription     :='0 Grad';
ST02_62_Y15.sInit.DampBothTime        :=200;
ST02_62_Y15.sInit.KindOfValve         :='2G';
ST02_62_Y15.sInit.MaxTime             :=2000;

(* Init ST02_DT_62_B11 Schwenkarm 1 0 Grad (ValveSensor) *)
ST02_DT_62_B11.sInit.InstName            :='ST02_DT_62_B11';
ST02_DT_62_B11.sInit.BitName            :='+62B11';
ST02_DT_62_B11.sInit.Description         :='Schwenkarm 1 0 Grad';
ST02_DT_62_B11.sInit.SensorType          :=sValveSensorType_WORK;

(* Init ST02_DT_61_B41 Schwenkarm 1 180 Grad (ValveSensor) *)
ST02_DT_61_B41.sInit.InstName            :='ST02_DT_61_B41';
ST02_DT_61_B41.sInit.BitName            :='+61B41';
ST02_DT_61_B41.sInit.Description         :='Schwenkarm 2 180 Grad';
ST02_DT_61_B41.sInit.SensorType          :=sValveSensorType_WORK;

(* Init ST02_62_Y4 Kamera Ausschleusen Bandstrecke (Valve) *)
ST02_62_Y4.sInit.InstName            :='ST02_62_Y4';
ST02_62_Y4.sInit.BitName            :='+62Y4';
ST02_62_Y4.sInit.Description         :='Kamera Ausschleusen';
ST02_62_Y4.sInit.HomePosDefine       :=HOME_ALWAYS;
ST02_62_Y4.sInit.InitDescription     :='GS';
ST02_62_Y4.sInit.WorkDescription     :='AS';
ST02_62_Y4.sInit.DampBothTime        :=200;
ST02_62_Y4.sInit.KindOfValve         :='2G';
ST02_62_Y4.sInit.MaxTime             :=4000;

(* Init ST02_FDB_54_B11 Kamera Ausschleusen Bandstrecke eingefahren (ValveSensor) *)
ST02_FDB_54_B11.sInit.InstName            :='ST02_FDB_54_B11';
ST02_FDB_54_B11.sInit.BitName            :='+54B11';
ST02_FDB_54_B11.sInit.Description         :='Kamera Ausschleusen';
ST02_FDB_54_B11.sInit.SensorType          :=sValveSensorType_INIT;

(* Init ST02_FDB_54_B21 Kamera Ausschleusen Bandstrecke ausgefahren (ValveSensor) *)
ST02_FDB_54_B21.sInit.InstName            :='ST02_FDB_54_B21';
ST02_FDB_54_B21.sInit.BitName            :='+54B21';
ST02_FDB_54_B21.sInit.Description         :='Kamera Ausschleusen';
ST02_FDB_54_B21.sInit.SensorType          :=sValveSensorType_WORK;



(*Init ST02_62_Y17 Schwenkarm 1 ISK Fixierung ein/ausfahren(Valve) *)
ST02_62_Y17.sInit.InstName            :='ST02_62_Y17';
ST02_62_Y17.sInit.BitName            :='+62_Y17';
ST02_62_Y17.sInit.Description         :='Iso 1 fiexieren';
ST02_62_Y17.sInit.HomePosDefine       :=HOME_ALWAYS;
ST02_62_Y17.sInit.InitDescription     :='GS';
ST02_62_Y17.sInit.WorkDescription     :='AS';
ST02_62_Y17.sInit.DampBothTime        :=200;
ST02_62_Y17.sInit.KindOfValve         :='2G';
ST02_62_Y17.sInit.MaxTime             :=4000;

(* Init ST02_S1_66_B11 Schwenkarm 1 ISK Fixierung GST (ValveSensor) *)
ST02_S1_66_B11.sInit.InstName            :='ST02_S1_66_B21';
ST02_S1_66_B11.sInit.BitName            :='+S1_66B11';
ST02_S1_66_B11.sInit.Description         :='Iso fixieren';
ST02_S1_66_B11.sInit.SensorType          :=sValveSensorType_INIT;

(* Init ST02_S1_66_B21 Schwenkarm 1 ISK Fixierung AST (ValveSensor) *)
ST02_S1_66_B21.sInit.InstName            :='ST02_S1_66_B21';
ST02_S1_66_B21.sInit.BitName            :='+S1_66B21';
ST02_S1_66_B21.sInit.Description         :='Iso fixieren';
ST02_S1_66_B21.sInit.SensorType          :=sValveSensorType_WORK;


(*Init ST02_62_Y18 Schwenkarm 2 ISK Fixierung ein/ausfahren(Valve) (Valve) *)
ST02_62_Y18.sInit.InstName            :='ST02_62_Y18';
ST02_62_Y18.sInit.BitName            :='+62_Y18';
ST02_62_Y18.sInit.Description         :='Iso 2 fiexieren';
ST02_62_Y18.sInit.HomePosDefine       :=HOME_ALWAYS;
ST02_62_Y18.sInit.InitDescription     :='GS';
ST02_62_Y18.sInit.WorkDescription     :='AS';
ST02_62_Y18.sInit.DampBothTime        :=200;
ST02_62_Y18.sInit.KindOfValve         :='2G';
ST02_62_Y18.sInit.MaxTime             :=4000;

(* Init ST02_S1_66_B31 Schwenkarm 2 ISK Fixierung GST (ValveSensor) *)
ST02_S1_66_B31.sInit.InstName            :='ST02_S1_66_B31';
ST02_S1_66_B31.sInit.BitName            :='S1_66B31';
ST02_S1_66_B31.sInit.Description         :='Iso fixieren';
ST02_S1_66_B31.sInit.SensorType          :=sValveSensorType_INIT;

(* Init ST02_S1_66_B41 Schwenkarm 2 ISK Fixierung AST (ValveSensor) *)
ST02_S1_66_B41.sInit.InstName            :='ST02_S1_66_B41';
ST02_S1_66_B41.sInit.BitName            :='S1_66_B41';
ST02_S1_66_B41.sInit.Description         :='Iso fixieren';
ST02_S1_66_B41.sInit.SensorType          :=sValveSensorType_WORK;


(* Init ST02_35Y01 Einschaltventil Hauptluft Tampondruckanlage (Valve) *)
ST02_35Y01.sInit.InstName          :='ST02_35Y01';
ST02_35Y01.sInit.BitName          :='+35Y01';
ST02_35Y01.sInit.Description       :='Hauptluft Tampondrucker';
ST02_35Y01.sInit.HomePosDefine     :=HOME_ALWAYS;
ST02_35Y01.sInit.InitDescription   :='GS';
ST02_35Y01.sInit.WorkDescription   :='AS';
ST02_35Y01.sInit.DampBothTime      :=0;
ST02_35Y01.sInit.MaxTime           :=2000;
ST02_35Y01.sInit.KindOfValve       :='A';
END_PROGRAM

(* POU Stations/ST_03_Ruestsaetze/ST_03__Init/ST03_Init, ST *)
PROGRAM ST03_Init


VAR


	sDigInVisu: BOOL;
END_VAR
(*INIT Aufrufe für Rüstsätze*)
Init_154polRP();	Init_154pol();
Init_160pol();		Init_206pol();
Init_92pol();		Init_124pol();
Init_46pol();		Init_NOX5_6pol();
Init_NOX4pol();	Init_88pol();
Init_7pol();		Init_88polAMG();
Init_120pol();		Init_21pol();
Init_191pol();		Init_48pol();
Init_72pol();		Init_268pol_102pol_neu();
Init_268polRP();	Init_33pol();

(* ----------------------------------------------------------------------------------------- *)
IF NOT MP.ST03.SGM_3621 THEN
	(*Init ST03_51_M1 Förderbandmotor*)
	ST03_51_M1.sConfig.Description		:='Förderband';
	ST03_51_M1.sConfig.InstName			:='ST03_51_M1';
	ST03_51_M1.sConfig.Aktiv				:=TRUE;
	ST03_51_M1.sConfig.Skalierfaktor		:=360.0 / (EXPT(2,20))	; (*360°/ 20 bit Encoder =0.00034332275390625*)
	ST03_51_M1.sConfig.Getriebefaktor		:=25;
	ST03_51_M1.sConfig.Modulo			:=FALSE;
	ST03_51_M1.sConfig.Pos_Faktor		:=157.07;			(*Weg bei einer Umdrehung in mm (nach Getriebe)*)
	ST03_51_M1.sConfig.maxRpm			:=5338;
	ST03_51_M1.sConfig.ModeOfOperation	:=CSP;				(*CSP,CSV,CST,CSTCA muss an der KLemme (Coe-Online 7010.03) eingestellt werden*)
	(*(CSP) position mode*)
	ST03_51_M1.sConfig.Torque_Limit		:=0;			(*bei 0 ausgeschaltet*)
	ST03_51_M1.sConfig.SW_Limit_on		:=FALSE;
	ST03_51_M1.sConfig.SW_Limit_min		:=-EXPT(2,32);
	ST03_51_M1.sConfig.SW_Limit_max		:=EXPT(2,32);
	ST03_51_M1.sConfig.lr_kp 				:= 800;
	ST03_51_M1.sConfig.lr_ki 				:= 100.0;
	ST03_51_M1.sConfig.lr_kd 				:= 50;
ELSE
	(* Init ST03_A5 Bandantrieb Förderbandmotor Oriental (nur 3621) Ein (DigOutIn)   ST08_170_K2 *)
	ST03_A5.sInit.InstName               :='ST03_A5';
	ST03_A5.sInit.Description            :='Förderbandmotor Isokörper';
	ST03_A5.sInit.BitOutName             :='-3_A5';
	ST03_A5.sInit.BitInName              :='';
	ST03_A5.sInit.HomePosOutput          :=2; (* 0: Signal=Low, 1: Signal=High, 2: always  *)
	ST03_A5.sInit.MaxTime                :=2000;
	ST03_A5.sInit.EnableInEveryMode  :=TRUE;
END_IF

(* Init ST03_V2 Störung Motor Förderband Oriental (DigIn) *)
ST03_V2.sInit.InstName               :='ST03_V2';
ST03_V2.sInit.Description            :='Störung Motor Förderband';
ST03_V2.sInit.BitInName              :='+3-V2';
ST03_V2.sInit.HomePosSignal          :=2; (* 0: Signal=Low, 1: Signal=High, 2: always  *)
ST03_V2.sInit.MaxTime                :=10;
ST03_V2.sInit.EnableInEveryMode       :=TRUE;

(* Init ST03_601V1_A1  Förderband Prüfteile (DigOutIn)  *)
ST03_601V1_A1.sInit.InstName               :='ST03_601V1_A1';
ST03_601V1_A1.sInit.Description            :='Förderband Prüfteile';
ST03_601V1_A1.sInit.BitOutName             :='-60V1_A1';
ST03_601V1_A1.sInit.BitInName              :='';
ST03_601V1_A1.sInit.HomePosOutput          :=2; (* 0: Signal=Low, 1: Signal=High, 2: always  *)
ST03_601V1_A1.sInit.MaxTime                :=2000;
ST03_601V1_A1.sInit.EnableInEveryMode  			:=TRUE;

(* ----------------------------------------------------------------------------------------- *)
(* 																	Roboter																									 *)
(* ----------------------------------------------------------------------------------------- *)
Visu.Robot01.TcpIpAdress:=MP.ST03.RobotIPAdress;
Robot01.sInit.InstName				:='Robot01';
Robot01.sInit.BitName				:='+3-125_A1';
Robot01.sInit.Description				:='ST03 Roboter';
Robot01.sInit.TcpIPAdress			:=MP.ST03.RobotIPAdress; (*10.16.55.130*)
Robot01.sInit.TcpIPSocket			:=2000;
Robot01.sInit.MaxTime				:=40000;
Robot01.sInit.WithToolHandling		:=TRUE;
Robot01.sInit.ToolMaxTime			:=2000;

(* Init ST03_125_F1 Absicherung Roboter iO (DigIn) *)
ST03_125_F1.sInit.InstName               :='ST03_125_F1';
ST03_125_F1.sInit.Description            :='Absicherung Roboter iO';
ST03_125_F1.sInit.BitInName              :='+3-125_F1';
ST03_125_F1.sInit.HomePosSignal          :=2; (* 0: Signal=Low, 1: Signal=High, 2: always  *)
ST03_125_F1.sInit.MaxTime                :=10;
ST03_125_F1.sInit.EnableInEveryMode       :=TRUE;

(* Init ST03_400_B12_6 Schwenkmodul GST (Roboterkopf) (DigIn) *)
ST03_400_B12_6.sInit.InstName           :='ST03_400_B12_6';
ST03_400_B12_6.sInit.Description        :='Rob. ST03 Schwenken GST';
ST03_400_B12_6.sInit.BitInName          :='+3-400_B12_6';
ST03_400_B12_6.sInit.HomePosSignal      :=2; (* 0: Signal=Low, 1: Signal=High, 2: always  *)
ST03_400_B12_6.sInit.MaxTime            :=2000;

(* Init ST03_400_B12_7 Schwenkmodul AST (Roboter) (DigIn) *)
ST03_400_B12_7.sInit.InstName           :='ST03_400_B12_7';
ST03_400_B12_7.sInit.Description        :='Rob. ST03 Schwenken AST';
ST03_400_B12_7.sInit.BitInName          :='+3-400_B12_7';
ST03_400_B12_7.sInit.HomePosSignal      :=2; (* 0: Signal=Low, 1: Signal=High, 2: always  *)
ST03_400_B12_7.sInit.MaxTime            :=2000;

(* Init St03_120_A1_A14 Rob. opt. Tool 2 ist Ein (DigIn) *)
St03_120_A1_A14.sInit.InstName           :='St03_120_A1_A14';
St03_120_A1_A14.sInit.Description        :='Rob. opt. Tool 2 ist Ein';
St03_120_A1_A14.sInit.BitInName          :='+3-120_A1_A14';
St03_120_A1_A14.sInit.HomePosSignal      :=2; (* 0: Signal=Low, 1: Signal=High, 2: always  *)
St03_120_A1_A14.sInit.MaxTime            :=2000;

(* Init ST03_BG3_S53_0 Start Band für Dummyprüfung (DigIn) *)
ST03_BG3_S53_0.sInit.InstName               :='ST03_BG3_S53_0';
ST03_BG3_S53_0.sInit.Description            :='Start Band für Dummyprüfung';
ST03_BG3_S53_0.sInit.BitInName              :='+0-BG3_S53_0';
ST03_BG3_S53_0.sInit.HomePosSignal          :=2; (* 0: Signal=Low, 1: Signal=High, 2: always  *)
ST03_BG3_S53_0.sInit.MaxTime                :=2000;
ST03_BG3_S53_0.sInit.EnableInEveryMode   	 :=TRUE;

(* Init ST03_BG3_X53_0 LED TasterStart Band für Dummyprüfung (DigOutIn) *)
ST03_BG3_X53_0.sInit.InstName          :='ST03_BG3_X53_0';
ST03_BG3_X53_0.sInit.Description       :='LED TasterStart Band für Dummyprüfung';
ST03_BG3_X53_0.sInit.BitOutName        :='+ST03_BG3_X53_0';
ST03_BG3_X53_0.sInit.BitInName         :='';
ST03_BG3_X53_0.sInit.HomePosSignal     :=2; (* 0: Signal=Low, 1: Signal=High, 2: always  *)
ST03_BG3_X53_0.sInit.MaxTime           :=2000;

(* Init ST03_400_B54_7 Tray Testteile in Position (DigIn) *)
ST03_400_B54_7.sInit.InstName            :='ST03_400_B54_7';
ST03_400_B54_7.sInit.Description         :='Tray Testteile in Position';
ST03_400_B54_7.sInit.BitInName           :='+8-400_B54.7';
ST03_400_B54_7.sInit.HomePosSignal       :=2; (* 0: Signal=Low, 1: Signal=High, 2: always  *)
ST03_400_B54_7.sInit.MaxTime             :=2000;

(* Init ST03_8_75_B13_5 voll/belegt keine Prüfteile mehr (DigIn) *)
ST03_8_75_B13_5.sInit.InstName            :='ST03_8_75_B13_5';
ST03_8_75_B13_5.sInit.Description         :='voll/belegt keine Prüfteile mehr';
ST03_8_75_B13_5.sInit.BitInName           :='+8-75_B13.5';
ST03_8_75_B13_5.sInit.HomePosSignal       :=2; (* 0: Signal=Low, 1: Signal=High, 2: always  *)
ST03_8_75_B13_5.sInit.MaxTime             :=2000;

(* Init ST03_8_75_B13_6 belegt mit 6 Prüfteile (DigIn) *)
ST03_8_75_B13_6.sInit.InstName            :='ST03_8_75_B13_6';
ST03_8_75_B13_6.sInit.Description         :='belegt mit 6 Prüfteile';
ST03_8_75_B13_6.sInit.BitInName           :='+8-75_B13.6';
ST03_8_75_B13_6.sInit.HomePosSignal       :=2; (* 0: Signal=Low, 1: Signal=High, 2: always  *)
ST03_8_75_B13_6.sInit.MaxTime             :=2000;

(* Init ST03_65_Q1 LED TasterStart Band für Dummyprüfung (DigOutIn) *)
ST03_65_Q1.sInit.InstName          :='ST03_65_Q1';
ST03_65_Q1.sInit.Description       :='Kühltunnel (Lüfter)';
ST03_65_Q1.sInit.BitOutName        :='+ST03_65_Q1';
ST03_65_Q1.sInit.BitInName         :='';
ST03_65_Q1.sInit.HomePosSignal     :=2; (* 0: Signal=Low, 1: Signal=High, 2: always  *)
ST03_65_Q1.sInit.MaxTime           :=2000;

(* Init ST03_65_F1 Tray Testteile in Position (DigIn) *)
ST03_65_F1.sInit.InstName            :='ST03_65_F1';
ST03_65_F1.sInit.Description         :='Sicherung Kühltunnel (Lüfter)';
ST03_65_F1.sInit.BitInName           :='+8-65_F1';
ST03_65_F1.sInit.HomePosSignal       :=2; (* 0: Signal=Low, 1: Signal=High, 2: always  *)
ST03_65_F1.sInit.MaxTime             :=2000;
END_PROGRAM
ACTION Init_120pol:
(*Rüstsatz 120 pol ==================================================================================*)

(* Init ST03_531_B69_0 Zuführung  frei zum Ablegen ISK SP Maschine (DigIn) *)
ST03_531_B69_0.sInit.InstName            :='ST03_531_B69_0';
ST03_531_B69_0.sInit.Description         :='frei zum Ablegen ISK SP Maschine';
ST03_531_B69_0.sInit.BitInName           :='+8-531_B69.0';
ST03_531_B69_0.sInit.HomePosSignal       :=2; (* 0: Signal=Low, 1: Signal=High, 2: always  *)
ST03_531_B69_0.sInit.MaxTime             :=2000;
ST03_531_B69_0.sInit.EnableInEveryMode   :=TRUE;

(* Init ST03_531_B69_1 Zuführung Vereinzler eingefahren GST (ValveSensor) *)
ST03_531_B69_1.sInit.InstName		:='ST03_531_B69_1';
ST03_531_B69_1.sInit.BitName		:='+8_531_B69.1';
ST03_531_B69_1.sInit.Description	:=' Vereinzler eingefahren GST';
ST03_531_B69_1.sInit.SensorType	:=sValveSensorType_INIT;

(* Init ST03_531_B69_2 Zuführung Vereinzler ausgefahren AST (ValveSensor) *)
ST03_531_B69_2.sInit.InstName		:='ST03_531_B69_2';
ST03_531_B69_2.sInit.BitName		:='+8_531_B69.2';
ST03_531_B69_2.sInit.Description	:=' Vereinzler ausgefahren AST';
ST03_531_B69_2.sInit.SensorType	:=sValveSensorType_WORK;

(* Init ST03_531_B69_3 Zuführung Stopper eingefahren AST (ValveSensor) *)
ST03_531_B69_3.sInit.InstName		:='ST03_531_B69_3';
ST03_531_B69_3.sInit.BitName		:='+8_531_B69.3';
ST03_531_B69_3.sInit.Description	:='Stopper eingefahren AST';
ST03_531_B69_3.sInit.SensorType	:=sValveSensorType_WORK;

(* Init ST03_531_B69_4 Zuführung Stopper ausgefahren GST (ValveSensor) *)
ST03_531_B69_4.sInit.InstName		:='ST03_531_B69_4';
ST03_531_B69_4.sInit.BitName		:='+8_531_B69.4';
ST03_531_B69_4.sInit.Description	:='Stopper ausgefahren GST';
ST03_531_B69_4.sInit.SensorType	:=sValveSensorType_INIT;;

(* Init ST03_531_B69_6 ISK anwesend am Stopper (DigIn) *)
ST03_531_B69_6.sInit.InstName            :='ST03_531_B69_6';
ST03_531_B69_6.sInit.Description         :='ISK anwesend am Stopper';
ST03_531_B69_6.sInit.BitInName           :='+8-531_B69.6';
ST03_531_B69_6.sInit.HomePosSignal       :=2; (* 0: Signal=Low, 1: Signal=High, 2: always  *)
ST03_531_B69_6.sInit.MaxTime             :=2000;
ST03_531_B69_6.sInit.EnableInEveryMode   :=TRUE;

(* Init ST03_531_B69_7 ISK rechts Lageerkennung (DigIn) *)
ST03_531_B69_7.sInit.InstName            :='ST03_531_B69_7';
ST03_531_B69_7.sInit.Description         :='ISK Lageerkennung rechts.';
ST03_531_B69_7.sInit.BitInName           :='+8-531_B69.7';
ST03_531_B69_7.sInit.HomePosSignal       :=2; (* 0: Signal=Low, 1: Signal=High, 2: always  *)
ST03_531_B69_7.sInit.MaxTime             :=2000;
ST03_531_B69_7.sInit.EnableInEveryMode   :=TRUE;

(* Init ST03_562_B70_0 ISK links Lageerkennung (DigIn) *)
ST03_532_B70_0.sInit.InstName            :='ST03_532_B70_0';
ST03_532_B70_0.sInit.Description         :='ISK Lageerkennung links';
ST03_532_B70_0.sInit.BitInName           :='+8-532_B70.0';
ST03_532_B70_0.sInit.HomePosSignal       :=2; (* 0: Signal=Low, 1: Signal=High, 2: always  *)
ST03_532_B70_0.sInit.MaxTime             :=2000;
ST03_532_B70_0.sInit.EnableInEveryMode   :=TRUE;

(* Init ST03_532_Y70_1   Zuführung  Vereinzler AST/GST (Valve) *)
ST03_532_Y70_1.sInit.InstName            :='ST03_532_Y70_1';
ST03_532_Y70_1.sInit.BitName            :='+8-532_Y70.1';
ST03_532_Y70_1.sInit.Description         :=' Zuführung Vereinzler AST/GST';
ST03_532_Y70_1.sInit.HomePosDefine       :=HOME_ALWAYS;
ST03_532_Y70_1.sInit.InitDescription     :='GS einfahren';
ST03_532_Y70_1.sInit.WorkDescription     :='AS ausfahren';
ST03_532_Y70_1.sInit.DampBothTime        :=200;
ST03_532_Y70_1.sInit.KindOfValve         :='A';
ST03_532_Y70_1.sInit.MaxTime             :=2000;

(* Init ST03_532_Y70_2   Zuführung  Stopper AST/GST (Valve) *)
ST03_532_Y70_2.sInit.InstName            :='ST03_532_Y70_2';
ST03_532_Y70_2.sInit.BitName            :='+8-532_Y70.2';
ST03_532_Y70_2.sInit.Description         :=' Zuführung Stopper AST/GST';
ST03_532_Y70_2.sInit.HomePosDefine       :=HOME_ALWAYS;
ST03_532_Y70_2.sInit.InitDescription     :='GS ausfahren';
ST03_532_Y70_2.sInit.WorkDescription     :='AS einfahren';
ST03_532_Y70_2.sInit.DampBothTime        :=200;
ST03_532_Y70_2.sInit.KindOfValve         :='A';
ST03_532_Y70_2.sInit.MaxTime             :=2000;
END_ACTION
ACTION Init_124pol:
(*========================= Rüstsatz 124 polig===============================*)

(* Init ST03_451_B69_0 Förderbandeinheit  Zuführung Vereinzler AST (ValveSensor) *)
ST03_451_B69_0.sInit.InstName            :='ST03_451_B69_0';
ST03_451_B69_0.sInit.BitName            :='+8_451_B69.0';
ST03_451_B69_0.sInit.Description         :='Förderbandeinheit  Zuführung Vereinzler AST';
ST03_451_B69_0.sInit.SensorType          :=sValveSensorType_INIT;

(* Init ST03_451_B69_1 Förderbandeinheit  Zuführung Vereinzler GST (ValveSensor) *)
ST03_451_B69_1.sInit.InstName            :='ST03_451_B69_1';
ST03_451_B69_1.sInit.BitName            :='+8_451_B69.1';
ST03_451_B69_1.sInit.Description         :='Förderbandeinheit  Zuführung Vereinzler GST';
ST03_451_B69_1.sInit.SensorType          :=sValveSensorType_WORK;

(* Init ST03_451_B69_2 Förderbandeinheit  Zuführung Stopper AST (ValveSensor) *)
ST03_451_B69_2.sInit.InstName            :='ST03_451_B69_2';
ST03_451_B69_2.sInit.BitName            :='+8_451_B69.2';
ST03_451_B69_2.sInit.Description         :='Förderband linke Zuführung Stopper AST';
ST03_451_B69_2.sInit.SensorType          :=sValveSensorType_INIT;

(* Init ST03_451_B69_3 Förderbandeinheit  Zuführung Stopper GST (ValveSensor) *)
ST03_451_B69_3.sInit.InstName            :='ST03_451_B69_3';
ST03_451_B69_3.sInit.BitName            :='+8_451_B69.3';
ST03_451_B69_3.sInit.Description         :='Förderband linke Zuführung Stopper GST';
ST03_451_B69_3.sInit.SensorType          :=sValveSensorType_WORK;

(* Init ST03_451_B69_4  Zuführung  frei zum Ablegen ISK SP Maschine Pos.1 (DigIn) *)
ST03_451_B69_4.sInit.InstName            :='ST03_451_B69_4';
ST03_451_B69_4.sInit.Description         :='Zuführung links frei zum Ablegen ISK SP Maschine Pos1';
ST03_451_B69_4.sInit.BitInName           :='+8-451_B69.4';
ST03_451_B69_4.sInit.HomePosSignal       :=2; (* 0: Signal=Low, 1: Signal=High, 2: always  *)
ST03_451_B69_4.sInit.MaxTime             :=2000;
ST03_451_B69_4.sInit.EnableInEveryMode   :=TRUE;

(* Init ST03_451_B69_7  ISK anwesend am Vereinzler (DigIn) *)
ST03_451_B69_7.sInit.InstName            :='ST03_451_B69_7';
ST03_451_B69_7.sInit.Description         :='ISK anwesend am Vereinzler';
ST03_451_B69_7.sInit.BitInName           :='+8-451_B69.7';
ST03_451_B69_7.sInit.HomePosSignal       :=2; (* 0: Signal=Low, 1: Signal=High, 2: always  *)
ST03_451_B69_7.sInit.MaxTime             :=2000;
ST03_451_B69_7.sInit.EnableInEveryMode   :=TRUE;

(* Init ST03_452_B70_1  Züführung  ISK Lageerkennung 1 (DigIn) *)
ST03_452_B70_1.sInit.InstName            :='ST03_452_B70_1';
ST03_452_B70_1.sInit.Description         :='Züführung  ISK Lageerkennung 1';
ST03_452_B70_1.sInit.BitInName           :='+8-452_B70.1';
ST03_452_B70_1.sInit.HomePosSignal       :=2; (* 0: Signal=Low, 1: Signal=High, 2: always  *)
ST03_452_B70_1.sInit.MaxTime             :=2000;
ST03_452_B70_1.sInit.EnableInEveryMode   :=TRUE;

(* Init ST03_452_B70_2  Züführung  ISK Lageerkennung 2 (DigIn) *)
ST03_452_B70_2.sInit.InstName            :='ST03_452_B70_2';
ST03_452_B70_2.sInit.Description         :='Züführung  ISK Lageerkennung 2';
ST03_452_B70_2.sInit.BitInName           :='+8-452_B70.2';
ST03_452_B70_2.sInit.HomePosSignal       :=2; (* 0: Signal=Low, 1: Signal=High, 2: always  *)
ST03_452_B70_2.sInit.MaxTime             :=2000;
ST03_452_B70_2.sInit.EnableInEveryMode   :=TRUE;

(* Init ST03_453_B70_4  ISK anwesend Übergabeposition Roboter (DigIn) *)
ST03_453_B70_4.sInit.InstName            :='ST03_453_B70_4';
ST03_453_B70_4.sInit.Description         :='Zuführung ISK auf Übergabeposition Robo Palettierer ';
ST03_453_B70_4.sInit.BitInName           :='+8-453_B70.4';
ST03_453_B70_4.sInit.HomePosSignal       :=2; (* 0: Signal=Low, 1: Signal=High, 2: always  *)
ST03_453_B70_4.sInit.MaxTime             :=2000;
ST03_453_B70_4.sInit.EnableInEveryMode   :=TRUE;

(* Init ST03_453_Y70_5 Förderband  Zuführung Vereinzler (Valve) *)
ST03_453_Y70_5.sInit.InstName            :='ST03_453_Y70_5';
ST03_453_Y70_5.sInit.BitName            :='+8-453_Y70.5';
ST03_453_Y70_5.sInit.Description         :='Förderband  Zuführung Vereinzler';
ST03_453_Y70_5.sInit.HomePosDefine       :=HOME_ALWAYS;
ST03_453_Y70_5.sInit.InitDescription     :='GS einfahren';
ST03_453_Y70_5.sInit.WorkDescription     :='AS ausfahren';
ST03_453_Y70_5.sInit.DampBothTime        :=200;
ST03_453_Y70_5.sInit.KindOfValve         :='A';
ST03_453_Y70_5.sInit.MaxTime             :=2000;

(* Init ST03_453_Y70_6 Förderband  Zuführung Stopper (Valve) *)
ST03_453_Y70_6.sInit.InstName            :='ST03_453_Y70_6';
ST03_453_Y70_6.sInit.BitName            :='+8-453_Y70.6';
ST03_453_Y70_6.sInit.Description         :='Förderband  Zuführung Stopper';
ST03_453_Y70_6.sInit.HomePosDefine       :=HOME_ALWAYS;
ST03_453_Y70_6.sInit.InitDescription     :='GS ausfahren';
ST03_453_Y70_6.sInit.WorkDescription     :='AS einfahren';
ST03_453_Y70_6.sInit.DampBothTime        :=200;
ST03_453_Y70_6.sInit.KindOfValve         :='A';
ST03_453_Y70_6.sInit.MaxTime             :=2000;
END_ACTION
ACTION Init_154pol:
(*Rüstsatz 154pol*)
(* Init ST03_425_B67_0 Förderbandeinheit  Zuführung Vereinzler AST (ValveSensor) *)
ST03_425_B67_0.sInit.InstName            :='ST03_425_B67_0';
ST03_425_B67_0.sInit.BitName            :='+8_425_B67.0';
ST03_425_B67_0.sInit.Description         :='Förderbandeinheit  Zuführung Vereinzler AST';
ST03_425_B67_0.sInit.SensorType          :=sValveSensorType_INIT;

(* Init ST03_425_B67_1 Förderbandeinheit  Zuführung Vereinzler GST (ValveSensor) *)
ST03_425_B67_1.sInit.InstName            :='ST03_425_B67_1';
ST03_425_B67_1.sInit.BitName            :='+8_425_B67.1';
ST03_425_B67_1.sInit.Description         :='Förderbandeinheit  Zuführung Vereinzler GST';
ST03_425_B67_1.sInit.SensorType          :=sValveSensorType_WORK;

(* Init ST03_425_B67_2 Förderbandeinheit  Zuführung Stopper AST (ValveSensor) *)
ST03_425_B67_2.sInit.InstName            :='ST03_425_B67_2';
ST03_425_B67_2.sInit.BitName            :='+8_425_B67.2';
ST03_425_B67_2.sInit.Description         :='Förderband linke Zuführung Stopper AST';
ST03_425_B67_2.sInit.SensorType          :=sValveSensorType_INIT;

(* Init ST03_425_B67_3 Förderbandeinheit  Zuführung Stopper GST (ValveSensor) *)
ST03_425_B67_3.sInit.InstName            :='ST03_425_B67_3';
ST03_425_B67_3.sInit.BitName            :='+8_425_B67.3';
ST03_425_B67_3.sInit.Description         :='Förderband linke Zuführung Stopper GST';
ST03_425_B67_3.sInit.SensorType          :=sValveSensorType_WORK;

(* Init ST03_425_B67_4  Zuführung  frei zum Ablegen ISK SP Maschine Pos.1 (DigIn) *)
ST03_425_B67_4.sInit.InstName            :='ST03_425_B67_4';
ST03_425_B67_4.sInit.Description         :='Zuführung links frei zum Ablegen ISK SP Maschine Pos1';
ST03_425_B67_4.sInit.BitInName           :='+8-425_B67.4';
ST03_425_B67_4.sInit.HomePosSignal       :=2; (* 0: Signal=Low, 1: Signal=High, 2: always  *)
ST03_425_B67_4.sInit.MaxTime             :=2000;
ST03_425_B67_4.sInit.EnableInEveryMode   :=TRUE;

(* Init ST03_425_B67_5  Zuführung  frei zum Ablegen ISK SP Maschine Pos.2 (DigIn) *)
ST03_425_B67_5.sInit.InstName            :='ST03_425_B67_5';
ST03_425_B67_5.sInit.Description         :='Zuführung links frei zum Ablegen ISK SP Maschine Pos2';
ST03_425_B67_5.sInit.BitInName           :='+8-425_B67.5';
ST03_425_B67_5.sInit.HomePosSignal       :=2; (* 0: Signal=Low, 1: Signal=High, 2: always  *)
ST03_425_B67_5.sInit.MaxTime             :=2000;
ST03_425_B67_5.sInit.EnableInEveryMode   :=TRUE;

(* Init ST03_425_B67_6  Zuführung  frei zum Ablegen ISK SP Maschine Pos.3 (DigIn) *)
ST03_425_B67_6.sInit.InstName            :='ST03_425_B67_6';
ST03_425_B67_6.sInit.Description         :='Zuführung links frei zum Ablegen ISK SP Maschine Pos3';
ST03_425_B67_6.sInit.BitInName           :='+8-425_B67.6';
ST03_425_B67_6.sInit.HomePosSignal       :=2; (* 0: Signal=Low, 1: Signal=High, 2: always  *)
ST03_425_B67_6.sInit.MaxTime             :=2000;
ST03_425_B67_6.sInit.EnableInEveryMode   :=TRUE;

(* Init ST03_425_B67_7  ISK anwesend am Vereinzler (DigIn) *)
ST03_425_B67_7.sInit.InstName            :='ST03_425_B67_7';
ST03_425_B67_7.sInit.Description         :='ISK anwesend am Vereinzler';
ST03_425_B67_7.sInit.BitInName           :='+8-425_B67.7';
ST03_425_B67_7.sInit.HomePosSignal       :=2; (* 0: Signal=Low, 1: Signal=High, 2: always  *)
ST03_425_B67_7.sInit.MaxTime             :=2000;
ST03_425_B67_7.sInit.EnableInEveryMode   :=TRUE;

(* Init ST03_426_B68_4  Züführung  ISK auf Übergabeposition Roboter Palettierer (DigIn) *)
ST03_426_B68_4.sInit.InstName            :='ST03_426_B68_4';
ST03_426_B68_4.sInit.Description         :='Züführung  ISK auf Übergabeposition Roboter Palettierer';
ST03_426_B68_4.sInit.BitInName           :='+8-426_B68.4';
ST03_426_B68_4.sInit.HomePosSignal       :=2; (* 0: Signal=Low, 1: Signal=High, 2: always  *)
ST03_426_B68_4.sInit.MaxTime             :=2000;
ST03_426_B68_4.sInit.EnableInEveryMode   :=TRUE;

(* Init ST03_426_Y68_5 Förderband  Zuführung Vereinzler (Valve) *)
ST03_426_Y68_5.sInit.InstName            :='ST03_426_Y68_5';
ST03_426_Y68_5.sInit.BitName            :='+8-426_Y68.5';
ST03_426_Y68_5.sInit.Description         :='Förderband  Zuführung Vereinzler';
ST03_426_Y68_5.sInit.HomePosDefine       :=HOME_ALWAYS;
ST03_426_Y68_5.sInit.InitDescription     :='GS einfahren';
ST03_426_Y68_5.sInit.WorkDescription     :='AS ausfahren';
ST03_426_Y68_5.sInit.DampBothTime        :=200;
ST03_426_Y68_5.sInit.KindOfValve         :='A';
ST03_426_Y68_5.sInit.MaxTime             :=2000;

(* Init ST03_426_Y68_6 Förderband  Zuführung Stopper (Valve) *)
ST03_426_Y68_6.sInit.InstName            :='ST03_426_Y68_6';
ST03_426_Y68_6.sInit.BitName            :='+8-426_Y68.6';
ST03_426_Y68_6.sInit.Description         :='Förderband  Zuführung Stopper';
ST03_426_Y68_6.sInit.HomePosDefine       :=HOME_ALWAYS;
ST03_426_Y68_6.sInit.InitDescription     :='GS ausfahren';
ST03_426_Y68_6.sInit.WorkDescription     :='AS einfahren';
ST03_426_Y68_6.sInit.DampBothTime        :=200;
ST03_426_Y68_6.sInit.KindOfValve         :='A';
ST03_426_Y68_6.sInit.MaxTime             :=2000;
END_ACTION
ACTION Init_154polRP:
(*Rüstsatz 154 Rasterplattel*)

(* Init ST03_418_B60_0 Förderband linke Zuführung Vereinzler AST  (ValveSensor) *)
ST03_418_B60_0.sInit.InstName            :='ST03_418_B60_0';
ST03_418_B60_0.sInit.BitName            :='+8_418_B60.0';
ST03_418_B60_0.sInit.Description         :='Förderband linke Zuführung Vereinzler AST';
ST03_418_B60_0.sInit.SensorType          :=sValveSensorType_WORK;

(* Init ST03_418_B60_1 Förderband linke Zuführung Vereinzler GST (ValveSensor) *)
ST03_418_B60_1.sInit.InstName            :='ST03_418_B60_1';
ST03_418_B60_1.sInit.BitName            :='+8_418_B60.1';
ST03_418_B60_1.sInit.Description         :='Förderband linke Zuführung Vereinzler GST';
ST03_418_B60_1.sInit.SensorType          :=sValveSensorType_INIT;

(* Init ST03_418_B60_2 Förderband rechte Zuführung Vereinzler AST (ValveSensor) *)
ST03_418_B60_2.sInit.InstName            :='ST03_418_B60_2';
ST03_418_B60_2.sInit.BitName            :='+8_418_B60.2';
ST03_418_B60_2.sInit.Description         :='Förderband rechte Zuführung Vereinzler AST';
ST03_418_B60_2.sInit.SensorType          :=sValveSensorType_WORK;

(* Init ST03_418_B60_3 Förderband rechte Zuführung Vereinzler GST(ValveSensor) *)
ST03_418_B60_3.sInit.InstName            :='ST03_418_B60_3';
ST03_418_B60_3.sInit.BitName            :='+8_418_B60.3';
ST03_418_B60_3.sInit.Description         :=' Förderband rechte Zuführung Vereinzler GST';
ST03_418_B60_3.sInit.SensorType          :=sValveSensorType_INIT;

(* Init ST03_418_B60_4 Förderband links/rechts Zuführung Stopper AST (ValveSensor) *)
ST03_418_B60_4.sInit.InstName            :='ST03_418_B60_4';
ST03_418_B60_4.sInit.BitName            :='+8_418_B60.4';
ST03_418_B60_4.sInit.Description         :='Förderband links/rechts Zuführung Stopper AST';
ST03_418_B60_4.sInit.SensorType          :=sValveSensorType_WORK;

(* Init ST03_418_B60_5 Förderband links/rechts Zuführung Stopper GST (ValveSensor) *)
ST03_418_B60_5.sInit.InstName            :='ST03_418_B60_5';
ST03_418_B60_5.sInit.BitName            :='+8_418_B60.5';
ST03_418_B60_5.sInit.Description         :='Förderband links/rechts Zuführung Stopper GST';
ST03_418_B60_5.sInit.SensorType          :=sValveSensorType_INIT;

(* Init ST03_418_B60_6 Zuführung links frei zum Ablegen ISK SP Maschine (DigIn) *)
ST03_418_B60_6.sInit.InstName            :='ST03_418_B60_6';
ST03_418_B60_6.sInit.Description         :='Zuführung links frei zum Ablegen ISK SP Maschine';
ST03_418_B60_6.sInit.BitInName           :='+8-418_B60.6';
ST03_418_B60_6.sInit.HomePosSignal       :=2; (* 0: Signal=Low, 1: Signal=High, 2: always  *)
ST03_418_B60_6.sInit.MaxTime             :=2000;
ST03_418_B60_6.sInit.EnableInEveryMode   :=TRUE;

(* Init ST03_418_B60_7 Zuführung rechts frei zum Ablegen ISK SP Maschine (DigIn) *)
ST03_418_B60_7.sInit.InstName            :='ST03_418_B60_7';
ST03_418_B60_7.sInit.Description         :='Zuführung rechts frei zum Ablegen ISK SP Maschine';
ST03_418_B60_7.sInit.BitInName           :='+8-418_B60.7';
ST03_418_B60_7.sInit.HomePosSignal       :=2; (* 0: Signal=Low, 1: Signal=High, 2: always  *)
ST03_418_B60_7.sInit.MaxTime             :=2000;
ST03_418_B60_7.sInit.EnableInEveryMode   :=TRUE;

(* Init ST03_419_B61_0 Förderband Zuführung links ISK anwesend zum Vereinzeln (DigIn) *)
ST03_419_B61_0.sInit.InstName            :='ST03_419_B61_0';
ST03_419_B61_0.sInit.Description         :='Förderband Zuführung links ISK anwesend zum Vereinzeln';
ST03_419_B61_0.sInit.BitInName           :='+8-419_B61.0';
ST03_419_B61_0.sInit.HomePosSignal       :=2; (* 0: Signal=Low, 1: Signal=High, 2: always  *)
ST03_419_B61_0.sInit.MaxTime             :=2000;
ST03_419_B61_0.sInit.EnableInEveryMode   :=TRUE;

(* Init ST03_419_B61_1 Förderband Zuführung rechts ISK anwesend zum Vereinzeln (DigIn) *)
ST03_419_B61_1.sInit.InstName            :='ST03_419_B61_1';
ST03_419_B61_1.sInit.Description         :='Förderband Zuführung rechts ISK anwesend zum Vereinzeln';
ST03_419_B61_1.sInit.BitInName           :='+8-419_B61.1';
ST03_419_B61_1.sInit.HomePosSignal       :=2; (* 0: Signal=Low, 1: Signal=High, 2: always  *)
ST03_419_B61_1.sInit.MaxTime             :=2000;
ST03_419_B61_1.sInit.EnableInEveryMode   :=TRUE;

(* Init ST03_419_B61_2 Züführung links ISK auf Übergabeposition Roboter Palettierer (DigIn) *)
ST03_419_B61_2.sInit.InstName            :='ST03_419_B61_2';
ST03_419_B61_2.sInit.Description         :='Züführung links ISK auf Übergabeposition Roboter Palettierer';
ST03_419_B61_2.sInit.BitInName           :='+8-419_B61.2';
ST03_419_B61_2.sInit.HomePosSignal       :=2; (* 0: Signal=Low, 1: Signal=High, 2: always  *)
ST03_419_B61_2.sInit.MaxTime             :=2000;
ST03_419_B61_2.sInit.EnableInEveryMode   :=TRUE;

(* Init ST03_419_B61_3 Züführung rechts ISK auf Übergabeposition Roboter Palettierer (DigIn) *)
ST03_419_B61_3.sInit.InstName            :='ST03_419_B61_3';
ST03_419_B61_3.sInit.Description         :='Züführung rechts ISK auf Übergabeposition Roboter Palettierer';
ST03_419_B61_3.sInit.BitInName           :='+8-419_B61.3';
ST03_419_B61_3.sInit.HomePosSignal       :=2; (* 0: Signal=Low, 1: Signal=High, 2: always  *)
ST03_419_B61_3.sInit.MaxTime             :=2000;
ST03_419_B61_3.sInit.EnableInEveryMode   :=TRUE;

(* Init ST03_419_Y61_5 Förderband linke Zuführung Vereinzler AST/GST (Valve) *)
ST03_419_Y61_5.sInit.InstName            :='ST03_419_Y61_5';
ST03_419_Y61_5.sInit.BitName            :='+8-419_Y61.5';
ST03_419_Y61_5.sInit.Description         :='Förderband linke Zuführung Vereinzler AST/GST';
ST03_419_Y61_5.sInit.HomePosDefine       :=HOME_ALWAYS;
ST03_419_Y61_5.sInit.InitDescription     :='GS einfahren';
ST03_419_Y61_5.sInit.WorkDescription     :='AS ausfahren';
ST03_419_Y61_5.sInit.DampBothTime        :=200;
ST03_419_Y61_5.sInit.KindOfValve         :='A';
ST03_419_Y61_5.sInit.MaxTime             :=2000;

(* Init ST03_419_Y61_6 Förderband rechte Zuführung Vereinzler AST/GST (Valve) *)
ST03_419_Y61_6.sInit.InstName            :='ST03_419_Y61_6';
ST03_419_Y61_6.sInit.BitName            :='+8-419_Y61.6';
ST03_419_Y61_6.sInit.Description         :='Förderband rechte Zuführung Vereinzler AST/GST';
ST03_419_Y61_6.sInit.HomePosDefine       :=HOME_ALWAYS;
ST03_419_Y61_6.sInit.InitDescription     :='GS einfahren';
ST03_419_Y61_6.sInit.WorkDescription     :='AS ausfahren';
ST03_419_Y61_6.sInit.DampBothTime        :=200;
ST03_419_Y61_6.sInit.KindOfValve         :='A';
ST03_419_Y61_6.sInit.MaxTime             :=2000;

(* Init ST03_419_Y61_7 Förderband links/rechts Züführung Stopper AST/GST (Valve) *)
ST03_419_Y61_7.sInit.InstName            :='ST03_419_Y61_7';
ST03_419_Y61_7.sInit.BitName            :='+8-419_Y61.7';
ST03_419_Y61_7.sInit.Description         :='Förderband links/rechts Züführung Stopper AST/GST';
ST03_419_Y61_7.sInit.HomePosDefine       :=HOME_ALWAYS;
ST03_419_Y61_7.sInit.InitDescription     :='GS ausfahren';
ST03_419_Y61_7.sInit.WorkDescription     :='AS einfahren';
ST03_419_Y61_7.sInit.DampBothTime        :=200;
ST03_419_Y61_7.sInit.KindOfValve         :='A';
ST03_419_Y61_7.sInit.MaxTime             :=2000;
END_ACTION
ACTION Init_160pol:
(*Rüstsatz 160pol*)
(* Init ST03_421_B63_0  Förderband Zuführung Vereinzler AST  (ValveSensor) *)
ST03_421_B63_0.sInit.InstName            :='ST03_421_B63_0';
ST03_421_B63_0.sInit.BitName            :='+8_421_B63.0';
ST03_421_B63_0.sInit.Description         :=' Förderband Zuführung Vereinzler AST';
ST03_421_B63_0.sInit.SensorType          :=sValveSensorType_WORK;

(* Init ST03_421_B63_1  Förderband Zuführung Vereinzler GST  (ValveSensor) *)
ST03_421_B63_1.sInit.InstName            :='ST03_421_B63_1';
ST03_421_B63_1.sInit.BitName            :='+8_421_B63.1';
ST03_421_B63_1.sInit.Description         :=' Förderband Zuführung Vereinzler GST';
ST03_421_B63_1.sInit.SensorType          :=sValveSensorType_INIT;

(* Init ST03_421_B63_2  Förderband Zuführung Stopper AST  (ValveSensor) *)
ST03_421_B63_2.sInit.InstName            :='ST03_421_B63_2';
ST03_421_B63_2.sInit.BitName            :='+8_421_B63.2';
ST03_421_B63_2.sInit.Description         :=' Förderband Zuführung Stopper AST';
ST03_421_B63_2.sInit.SensorType          :=sValveSensorType_INIT;

(* Init ST03_421_B63_3  Förderband Zuführung Stopper GST  (ValveSensor) *)
ST03_421_B63_3.sInit.InstName            :='ST03_421_B63_3';
ST03_421_B63_3.sInit.BitName            :='+8_421_B63.3';
ST03_421_B63_3.sInit.Description         :=' Förderband Zuführung Stopper GST';
ST03_421_B63_3.sInit.SensorType          :=sValveSensorType_WORK;

(* Init ST03_421_B63_4 Förderband frei zum Ablegen ISK SP Maschine Pos1 (DigIn) *)
ST03_421_B63_4.sInit.InstName            :='ST03_421_B63_4';
ST03_421_B63_4.sInit.Description         :='Förderband frei zum Ablegen ISK SP Maschine Pos1';
ST03_421_B63_4.sInit.BitInName           :='+8-421_B63.4';
ST03_421_B63_4.sInit.HomePosSignal       :=2; (* 0: Signal=Low, 1: Signal=High, 2: always  *)
ST03_421_B63_4.sInit.MaxTime             :=2000;
ST03_421_B63_4.sInit.EnableInEveryMode   :=TRUE;

(* Init ST03_421_B63_5 Förderband frei zum Ablegen ISK SP Maschine Pos2 (DigIn) *)
ST03_421_B63_5.sInit.InstName            :='ST03_421_B63_5';
ST03_421_B63_5.sInit.Description         :='Förderband frei zum Ablegen ISK SP Maschine Pos2';
ST03_421_B63_5.sInit.BitInName           :='+8-421_B63.5';
ST03_421_B63_5.sInit.HomePosSignal       :=2; (* 0: Signal=Low, 1: Signal=High, 2: always  *)
ST03_421_B63_5.sInit.MaxTime             :=2000;
ST03_421_B63_5.sInit.EnableInEveryMode   :=TRUE;

(* Init ST03_421_B63_6 Förderband frei zum Ablegen ISK SP Maschine Pos3 (DigIn) *)
ST03_421_B63_6.sInit.InstName            :='ST03_421_B63_6';
ST03_421_B63_6.sInit.Description         :='Förderband frei zum Ablegen ISK SP Maschine Pos3';
ST03_421_B63_6.sInit.BitInName           :='+8-421_B63.6';
ST03_421_B63_6.sInit.HomePosSignal       :=2; (* 0: Signal=Low, 1: Signal=High, 2: always  *)
ST03_421_B63_6.sInit.MaxTime             :=2000;
ST03_421_B63_6.sInit.EnableInEveryMode   :=TRUE;

(* Init ST03_421_B63_7 ISK anwesend am Vereinzler (DigIn) *)
ST03_421_B63_7.sInit.InstName            :='ST03_421_B63_7';
ST03_421_B63_7.sInit.Description         :='ISK anwesend am Vereinzler';
ST03_421_B63_7.sInit.BitInName           :='+8-421_B63.7';
ST03_421_B63_7.sInit.HomePosSignal       :=2; (* 0: Signal=Low, 1: Signal=High, 2: always  *)
ST03_421_B63_7.sInit.MaxTime             :=2000;
ST03_421_B63_7.sInit.EnableInEveryMode   :=TRUE;

(* Init ST03_422_B64_0 Förderband Trigger Tintenstrahldrucker 1 Rüstsatz (Lichtschranke) (DigIn) *)
ST03_422_B64_0.sInit.InstName            :='ST03_421_B64_0';
ST03_422_B64_0.sInit.Description         :='Förderband Trigger Tintenstrahldrucker (Lichtschranke)';
ST03_422_B64_0.sInit.BitInName           :='+8-421_B64.0';
ST03_422_B64_0.sInit.HomePosSignal       :=2; (* 0: Signal=Low, 1: Signal=High, 2: always  *)
ST03_422_B64_0.sInit.MaxTime             :=2000;
ST03_422_B64_0.sInit.EnableInEveryMode   :=TRUE;

(* Init ST03_423_B63_0 Förderband Trigger Tintenstrahldrucker 2 Rüstsatz (Lichtschranke) (DigIn) *)
ST03_423_B66_0.sInit.InstName            :='ST03_423_B66_0';
ST03_423_B66_0.sInit.Description         :='Förderband Trigger Tintenstrahldrucker (Lichtschranke)';
ST03_423_B66_0.sInit.BitInName           :='+8-423_B66.0';
ST03_423_B66_0.sInit.HomePosSignal       :=2; (* 0: Signal=Low, 1: Signal=High, 2: always  *)
ST03_423_B66_0.sInit.MaxTime             :=2000;
ST03_423_B66_0.sInit.EnableInEveryMode   :=TRUE;

(* Init ST03_8_B76_1 Förderband Trigger Tintenstrahldrucker (Lichtschranke) (DigIn) 3621 *)
ST03_8_B76_1.sInit.InstName            :='ST03_8_B76_1';
ST03_8_B76_1.sInit.Description         :='Förderband Trigger Tintenstrahldrucker (Lichtschranke)';
ST03_8_B76_1.sInit.BitInName           :='+8-B76_1';
ST03_8_B76_1.sInit.HomePosSignal       :=2; (* 0: Signal=Low, 1: Signal=High, 2: always  *)
ST03_8_B76_1.sInit.MaxTime             :=2000;
ST03_8_B76_1.sInit.EnableInEveryMode   :=TRUE;

(* Init ST03_8_B76_2 Förderband Trigger Tintenstrahldrucker (Lichtschranke) (DigIn) 3621 *)
ST03_8_B76_2.sInit.InstName            :='ST03_8_B76_2';
ST03_8_B76_2.sInit.Description         :='Förderband Trigger Tintenstrahldrucker (Lichtschranke)';
ST03_8_B76_2.sInit.BitInName           :='+8-B76_2';
ST03_8_B76_2.sInit.HomePosSignal       :=2; (* 0: Signal=Low, 1: Signal=High, 2: always  *)
ST03_8_B76_2.sInit.MaxTime             :=2000;
ST03_8_B76_2.sInit.EnableInEveryMode   :=TRUE;

(* Init ST03_422_B64_1  Förderband Zuführung Stopper 1 Kamera AST  (ValveSensor) *)
ST03_422_B64_1.sInit.InstName            :='ST03_422_B64_1';
ST03_422_B64_1.sInit.BitName            :='+8_422_B64.1';
ST03_422_B64_1.sInit.Description         :=' Förderband Zuführung Stopper Kamera AST';
ST03_422_B64_1.sInit.SensorType          :=sValveSensorType_WORK;

(* Init ST03_422_B64_2  Förderband Zuführung Stopper 1 Kamera GST  (ValveSensor) *)
ST03_422_B64_2.sInit.InstName            :='ST03_422_B64_2';
ST03_422_B64_2.sInit.BitName            :='+8_422_B64.2';
ST03_422_B64_2.sInit.Description         :=' Förderband Zuführung Stopper 1 Kamera GST';
ST03_422_B64_2.sInit.SensorType          :=sValveSensorType_INIT;

(* Init ST03_422_B64_3  Förderband ISK anwesend am Stopper 1 Kamera (DigIn) *)
ST03_422_B64_3.sInit.InstName            :='ST03_421_B64_3';
ST03_422_B64_3.sInit.Description         :=' Förderband ISK anwesend Stopper 1 Kamera';
ST03_422_B64_3.sInit.BitInName           :='+8-421_B64.3';
ST03_422_B64_3.sInit.HomePosSignal       :=2; (* 0: Signal=Low, 1: Signal=High, 2: always  *)
ST03_422_B64_3.sInit.MaxTime             :=2000;
ST03_422_B64_3.sInit.EnableInEveryMode   :=TRUE;

(* Init ST03_423_B65_0  Förderband Zuführung Stopper 2 Kamera AST  (ValveSensor) *)
ST03_423_B65_0.sInit.InstName            :='ST03_423_B65_0';
ST03_423_B65_0.sInit.BitName            :='+8_423_B65.0';
ST03_423_B65_0.sInit.Description         :=' Förderband Zuführung Stopper 2 Kamera AST';
ST03_423_B65_0.sInit.SensorType          :=sValveSensorType_WORK;

(* Init ST03_423_B65_1  Förderband Zuführung Stopper 2 Kamera GST  (ValveSensor) *)
ST03_423_B65_1.sInit.InstName            :='ST03_423_B65_1';
ST03_423_B65_1.sInit.BitName            :='+8_423_B65.1';
ST03_423_B65_1.sInit.Description         :=' Förderband Zuführung Stopper 2 Kamera GST';
ST03_423_B65_1.sInit.SensorType          :=sValveSensorType_INIT;

(* Init ST03_423_B65_2  Förderband ISK anwesend am Stopper 2 Kamera (DigIn) *)
ST03_423_B65_2.sInit.InstName            :='ST03_423_B65_2';
ST03_423_B65_2.sInit.Description         :=' Förderband ISK anwesend Stopper Kamera';
ST03_423_B65_2.sInit.BitInName           :='+8-423_B65.2';
ST03_423_B65_2.sInit.HomePosSignal       :=2; (* 0: Signal=Low, 1: Signal=High, 2: always  *)
ST03_423_B65_2.sInit.MaxTime             :=2000;
ST03_423_B65_2.sInit.EnableInEveryMode   :=TRUE;

(* Init ST03_423_B65_3  Förderband Zuführung Stopper 3 Kamera AST  (ValveSensor) *)
ST03_423_B65_3.sInit.InstName            :='ST03_423_B65_3';
ST03_423_B65_3.sInit.BitName            :='+8_423_B65.3';
ST03_423_B65_3.sInit.Description         :=' Förderband Zuführung Stopper 3 Kamera AST';
ST03_423_B65_3.sInit.SensorType          :=sValveSensorType_WORK;

(* Init ST03_423_B65_4  Förderband Zuführung Stopper 3 Kamera GST  (ValveSensor) *)
ST03_423_B65_4.sInit.InstName            :='ST03_423_B65_4';
ST03_423_B65_4.sInit.BitName            :='+8_423_B65.4';
ST03_423_B65_4.sInit.Description         :=' Förderband Zuführung Stopper 3 Kamera GST';
ST03_423_B65_4.sInit.SensorType          :=sValveSensorType_INIT;

(* Init ST03_423_B65_5  Förderband ISK anwesend am Stopper 3 Kamera (DigIn) *)
ST03_423_B65_5.sInit.InstName            :='ST03_423_B65_5';
ST03_423_B65_5.sInit.Description         :=' Förderband ISK anwesend Stopper Kamera';
ST03_423_B65_5.sInit.BitInName           :='+8-423_B65.5';
ST03_423_B65_5.sInit.HomePosSignal       :=2; (* 0: Signal=Low, 1: Signal=High, 2: always  *)
ST03_423_B65_5.sInit.MaxTime             :=2000;
ST03_423_B65_5.sInit.EnableInEveryMode   :=TRUE;

(* Init ST03_422_B64_4 Zuführung ISK auf Übergabeposition Robo Palettierer (DigIn) *)
ST03_422_B64_4.sInit.InstName            :='ST03_421_B64_4';
ST03_422_B64_4.sInit.Description         :='Zuführung ISK auf Übergabeposition Robo Palettierer';
ST03_422_B64_4.sInit.BitInName           :='+8-421_B64.4';
ST03_422_B64_4.sInit.HomePosSignal       :=2; (* 0: Signal=Low, 1: Signal=High, 2: always  *)
ST03_422_B64_4.sInit.MaxTime             :=2000;
ST03_422_B64_4.sInit.EnableInEveryMode   :=TRUE;

(* Init ST03_422_Y64_5 Förderband  Zuführung Vereinzler AST/GST (Valve) *)
ST03_422_Y64_5.sInit.InstName            :='ST03_422_Y64_5';
ST03_422_Y64_5.sInit.BitName            :='+8-419_Y64.5';
ST03_422_Y64_5.sInit.Description         :='Förderband  Zuführung Vereinzler AST/GST';
ST03_422_Y64_5.sInit.HomePosDefine       :=HOME_ALWAYS;
ST03_422_Y64_5.sInit.InitDescription     :='GS einfahren';
ST03_422_Y64_5.sInit.WorkDescription     :='AS ausfahren';
ST03_422_Y64_5.sInit.DampBothTime        :=200;
ST03_422_Y64_5.sInit.KindOfValve         :='A';
ST03_422_Y64_5.sInit.MaxTime             :=2000;

(* Init ST03_422_Y64_6 Förderband  Stopper Vereinzler AST/GST (Valve) *)
ST03_422_Y64_6.sInit.InstName            :='ST03_422_Y64_6';
ST03_422_Y64_6.sInit.BitName            :='+8-419_Y64.6';
ST03_422_Y64_6.sInit.Description         :='Förderband  Stopper Vereinzler AST/GST';
ST03_422_Y64_6.sInit.HomePosDefine       :=HOME_ALWAYS;
ST03_422_Y64_6.sInit.InitDescription     :='GS ausfahren';
ST03_422_Y64_6.sInit.WorkDescription     :='AS einfahren';
ST03_422_Y64_6.sInit.DampBothTime        :=200;
ST03_422_Y64_6.sInit.KindOfValve         :='A';
ST03_422_Y64_6.sInit.MaxTime             :=2000;

(* Init ST03_422_Y64_7 Förderband  Stopper 1 Kamera AST/GST (Valve) *)
ST03_422_Y64_7.sInit.InstName            :='ST03_422_Y64_7';
ST03_422_Y64_7.sInit.BitName            :='+8-419_Y64.7';
ST03_422_Y64_7.sInit.Description         :='Förderband  Stopper Kamera AST/GST';
ST03_422_Y64_7.sInit.HomePosDefine       :=HOME_ALWAYS;
ST03_422_Y64_7.sInit.InitDescription     :='GS ausfahren';
ST03_422_Y64_7.sInit.WorkDescription     :='AS einfahren';
ST03_422_Y64_7.sInit.DampBothTime        :=200;
ST03_422_Y64_7.sInit.KindOfValve         :='A';
ST03_422_Y64_7.sInit.MaxTime             :=2000;

(* Init ST03_423_Y65_6 Förderband  Stopper 2 Kamera AST/GST (Valve) *)
ST03_423_Y65_6.sInit.InstName            :='ST03_423_Y65_6';
ST03_423_Y65_6.sInit.BitName            :='+8-423_Y65.6';
ST03_423_Y65_6.sInit.Description         :='Förderband  Stopper Kamera AST/GST';
ST03_423_Y65_6.sInit.HomePosDefine       :=HOME_ALWAYS;
ST03_423_Y65_6.sInit.InitDescription     :='GS ausfahren';
ST03_423_Y65_6.sInit.WorkDescription     :='AS einfahren';
ST03_423_Y65_6.sInit.DampBothTime        :=200;
ST03_423_Y65_6.sInit.KindOfValve         :='2G';
ST03_423_Y65_6.sInit.MaxTime             :=2000;

(* Init ST03_423_Y65_7 Förderband  Stopper 3 Kamera AST/GST (Valve) *)
ST03_423_Y65_7.sInit.InstName            :='ST03_423_Y65_7';
ST03_423_Y65_7.sInit.BitName            :='+8-423_Y65.7';
ST03_423_Y65_7.sInit.Description         :='Förderband  Stopper Kamera AST/GST';
ST03_423_Y65_7.sInit.HomePosDefine       :=HOME_ALWAYS;
ST03_423_Y65_7.sInit.InitDescription     :='GS ausfahren';
ST03_423_Y65_7.sInit.WorkDescription     :='AS einfahren';
ST03_423_Y65_7.sInit.DampBothTime        :=200;
ST03_423_Y65_7.sInit.KindOfValve         :='2G';
ST03_423_Y65_7.sInit.MaxTime             :=2000;

(* Init ST03_33F4 Steckdosen Tintenstrahldrucker (DigIn) *)
ST03_33F4.sInit.InstName            :='ST03_33_F4';
ST03_33F4.sInit.Description         :='SteckdosenTintenstrahldrucker';
ST03_33F4.sInit.BitInName           :='+33_F4';
ST03_33F4.sInit.HomePosSignal       :=2; (* 0: Signal=Low, 1: Signal=High, 2: always  *)
ST03_33F4.sInit.MaxTime             :=2000;
ST03_33F4.sInit.EnableInEveryMode   :=TRUE;

(* Init ST03_70U3_1 Bereit/ Im Druck Tintenstrahldrucker Frontseite (DigIn) *)
ST03_70U3_1.sInit.InstName            :='ST03_70U3_1';
ST03_70U3_1.sInit.Description         :='Bereit/ Im Druck Frontseite';
ST03_70U3_1.sInit.BitInName           :='+70U3_1';
ST03_70U3_1.sInit.HomePosSignal       :=2; (* 0: Signal=Low, 1: Signal=High, 2: always  *)
ST03_70U3_1.sInit.MaxTime             :=2000;
ST03_70U3_1.sInit.EnableInEveryMode   :=TRUE;

(* Init ST03_70U3_2 Tank voll Tintenstrahldrucker Frontseite (DigIn) *)
ST03_70U3_2.sInit.InstName            :='ST03_70U3_2';
ST03_70U3_2.sInit.Description         :='Tank voll Drucker Frontseite';
ST03_70U3_2.sInit.BitInName           :='+70U3_2';
ST03_70U3_2.sInit.HomePosSignal       :=2; (* 0: Signal=Low, 1: Signal=High, 2: always  *)
ST03_70U3_2.sInit.MaxTime             :=2000;
ST03_70U3_2.sInit.EnableInEveryMode   :=TRUE;

(* Init ST03_70U3_3 Fehler/Störung Tintenstrahldrucker Frontseite (DigIn) *)
ST03_70U3_3.sInit.InstName            :='ST03_70U3_3';
ST03_70U3_3.sInit.Description         :='Fehler Drucker Frontseite';
ST03_70U3_3.sInit.BitInName           :='+70U3_3';
ST03_70U3_3.sInit.HomePosSignal       :=2; (* 0: Signal=Low, 1: Signal=High, 2: always  *)
ST03_70U3_3.sInit.MaxTime             :=2000;
ST03_70U3_3.sInit.EnableInEveryMode   :=TRUE;

(* Init ST03_71U3_1 Bereit/ Im Druck Tintenstrahldrucker Rückseite (DigIn) *)
ST03_71U3_1.sInit.InstName            :='ST03_71U3_1';
ST03_71U3_1.sInit.Description         :='Bereit/ Im Druck  Rückseite';
ST03_71U3_1.sInit.BitInName           :='+71U3_1';
ST03_71U3_1.sInit.HomePosSignal       :=2; (* 0: Signal=Low, 1: Signal=High, 2: always  *)
ST03_71U3_1.sInit.MaxTime             :=2000;
ST03_71U3_1.sInit.EnableInEveryMode   :=TRUE;

(* Init ST03_71U3_2 Tank voll Tintenstrahldrucker Rückseite (DigIn) *)
ST03_71U3_2.sInit.InstName            :='ST03_71U3_2';
ST03_71U3_2.sInit.Description         :='Tank voll Drucker Rückseite';
ST03_71U3_2.sInit.BitInName           :='+71U3_2';
ST03_71U3_2.sInit.HomePosSignal       :=2; (* 0: Signal=Low, 1: Signal=High, 2: always  *)
ST03_71U3_2.sInit.MaxTime             :=2000;
ST03_71U3_2.sInit.EnableInEveryMode   :=TRUE;

(* Init ST03_71U3_3 Steckdosenleise (DigIn) *)
ST03_71U3_3.sInit.InstName            :='ST03_71U3_3';
ST03_71U3_3.sInit.Description         :='Fehler Drucker Rückseite';
ST03_71U3_3.sInit.BitInName           :='+71U3_3';
ST03_71U3_3.sInit.HomePosSignal       :=2; (* 0: Signal=Low, 1: Signal=High, 2: always  *)
ST03_71U3_3.sInit.MaxTime             :=2000;
ST03_71U3_3.sInit.EnableInEveryMode   :=TRUE;

(* Init ST03_PLAN_70V1_1 Start  Bedrucken Tintenstrahldrucker Frontseite (DigOutIn) *)
ST03_PLAN_70V1_1.sInit.InstName               :='ST03_PLAN_70V1_1';
ST03_PLAN_70V1_1.sInit.Description            :='Start  Drucker Frontseite';
ST03_PLAN_70V1_1.sInit.BitOutName             :='+PLAN_70V1_1';
ST03_PLAN_70V1_1.sInit.BitInName              :='';
ST03_PLAN_70V1_1.sInit.HomePosOutput          :=2; (* 0: Signal=Low, 1: Signal=High, 2: always  *)
ST03_PLAN_70V1_1.sInit.MaxTime                :=2000;
ST03_PLAN_70V1_1.sInit.EnableInEveryMode  :=TRUE;

(* Init ST03_PLAN_71V1_2 Start  Bedrucken Tintenstrahldrucker Rückseite (DigOutIn) *)
ST03_PLAN_71V1_2.sInit.InstName               :='ST03_PLAN_71V1_2';
ST03_PLAN_71V1_2.sInit.Description            :='Start  Drucker Rückseite';
ST03_PLAN_71V1_2.sInit.BitOutName             :='+PLAN_71V1_2';
ST03_PLAN_71V1_2.sInit.BitInName              :='';
ST03_PLAN_71V1_2.sInit.HomePosOutput          :=2; (* 0: Signal=Low, 1: Signal=High, 2: always  *)
ST03_PLAN_71V1_2.sInit.MaxTime                :=2000;
ST03_PLAN_71V1_2.sInit.EnableInEveryMode  :=TRUE;

(* Init ST03_Y01 Einschaltventil Hauptluft Tintenstrahldrucker (Valve) *)
ST03_Y01.sInit.InstName          :='ST03_Y01';
ST03_Y01.sInit.InstName          :='+Y01';
ST03_Y01.sInit.Description       :='Hauptluft Tintenstrahldrucker';
ST03_Y01.sInit.HomePosDefine     :=HOME_ALWAYS;
ST03_Y01.sInit.InitDescription   :='ON';
ST03_Y01.sInit.WorkDescription   :='OFF';
ST03_Y01.sInit.DampBothTime      :=0;
ST03_Y01.sInit.MaxTime           :=2000;
ST03_Y01.sInit.KindOfValve       :='A';

(* Init ST03_S18 ST02 Druckschalter Wartungseinheit Hauptluft Tintenstrahldrucker min.6 bar (DigIn) ST02_35_S31*)
ST03_S18.sInit.InstName            :='ST03_S18';
ST03_S18.sInit.Description         :='ST02 Druckschalter Wartungseinheit Hauptluft min.6 bar';
ST03_S18.sInit.BitInName           :='-ST03_S18';
ST03_S18.sInit.HomePosSignal       :=2; (* 0: Signal=Low, 1: Signal=High, 2: always  *)
ST03_S18.sInit.MaxTime             :=2000;
ST03_S18.sInit.EnableInEveryMode   :=TRUE;

(* Init ST03_H6 Signalsäule GR Bedruckung IO (DigOutIn) *)
ST03_H6.sInit.InstName               :='ST03_H6';
ST03_H6.sInit.Description            :='Signalsäule GR Bedruckung IO';
ST03_H6.sInit.BitOutName             :='-H6';
ST03_H6.sInit.BitInName              :='';
ST03_H6.sInit.HomePosOutput          :=2; (* 0: Signal=Low, 1: Signal=High, 2: always  *)
ST03_H6.sInit.MaxTime                :=2000;
ST03_H6.sInit.EnableInEveryMode   	 :=TRUE;

(* Init ST03_H7 Signalsäule RD Sammelstörung Bedruckung (DigOutIn) *)
ST03_H7.sInit.InstName               :='ST03_H7';
ST03_H7.sInit.Description            :='Signalsäule GR Bedruckung IO';
ST03_H7.sInit.BitOutName             :='-H7';
ST03_H7.sInit.BitInName              :='';
ST03_H7.sInit.HomePosOutput          :=2; (* 0: Signal=Low, 1: Signal=High, 2: always  *)
ST03_H7.sInit.MaxTime                :=2000;
ST03_H7.sInit.EnableInEveryMode   	 :=TRUE;
END_ACTION
ACTION Init_191pol:
(*Rüstsatz 191 pol ==================================================================================*)

(* Init ST03_541_B69_0 Zuführung  frei zum Ablegen ISK SP Maschine (DigIn) *)
ST03_541_B69_0.sInit.InstName            :='ST03_541_B69_0';
ST03_541_B69_0.sInit.Description         :='frei zum Ablegen ISK SP Maschine';
ST03_541_B69_0.sInit.BitInName           :='+8-541_B69.0';
ST03_541_B69_0.sInit.HomePosSignal       :=2; (* 0: Signal=Low, 1: Signal=High, 2: always  *)
ST03_541_B69_0.sInit.MaxTime             :=2000;
ST03_541_B69_0.sInit.EnableInEveryMode   :=TRUE;

(* Init ST03_541_B69_1 Zuführung Vereinzler eingefahren GST (ValveSensor) *)
ST03_541_B69_1.sInit.InstName		:='ST03_541_B69_1';
ST03_541_B69_1.sInit.BitName		:='+8_541_B69.1';
ST03_541_B69_1.sInit.Description	:=' Vereinzler eingefahren GST';
ST03_541_B69_1.sInit.SensorType	:=sValveSensorType_INIT;

(* Init ST03_541_B69_2 Zuführung Vereinzler ausgefahren AST (ValveSensor) *)
ST03_541_B69_2.sInit.InstName		:='ST03_541_B69_2';
ST03_541_B69_2.sInit.BitName		:='+8_541_B69.2';
ST03_541_B69_2.sInit.Description	:=' Vereinzler ausgefahren AST';
ST03_541_B69_2.sInit.SensorType	:=sValveSensorType_WORK;

(* Init ST03_541_B69_3 Zuführung Stopper eingefahren AST (ValveSensor) *)
ST03_541_B69_3.sInit.InstName		:='ST03_541_B69_3';
ST03_541_B69_3.sInit.BitName		:='+8_541_B69.3';
ST03_541_B69_3.sInit.Description	:='Stopper eingefahren AST';
ST03_541_B69_3.sInit.SensorType	:=sValveSensorType_WORK;

(* Init ST03_541_B69_4 Zuführung Stopper ausgefahren GST (ValveSensor) *)
ST03_541_B69_4.sInit.InstName		:='ST03_541_B69_4';
ST03_541_B69_4.sInit.BitName		:='+8_541_B69.4';
ST03_541_B69_4.sInit.Description	:='Stopper ausgefahren GST';
ST03_541_B69_4.sInit.SensorType	:=sValveSensorType_INIT;;

(* Init ST03_541_B69_6 ISK anwesend am Stopper (DigIn) *)
ST03_541_B69_6.sInit.InstName            :='ST03_541_B69_6';
ST03_541_B69_6.sInit.Description         :='ISK anwesend am Stopper';
ST03_541_B69_6.sInit.BitInName           :='+8-541_B69.6';
ST03_541_B69_6.sInit.HomePosSignal       :=2; (* 0: Signal=Low, 1: Signal=High, 2: always  *)
ST03_541_B69_6.sInit.MaxTime             :=2000;
ST03_541_B69_6.sInit.EnableInEveryMode   :=TRUE;

(* Init ST03_541_B69_7 ISK links Lageerkennung (DigIn) *)
ST03_541_B69_7.sInit.InstName            :='ST03_541_B69_7';
ST03_541_B69_7.sInit.Description         :='ISK links Lageerkennung.';
ST03_541_B69_7.sInit.BitInName           :='+8-541_B69.7';
ST03_541_B69_7.sInit.HomePosSignal       :=2; (* 0: Signal=Low, 1: Signal=High, 2: always  *)
ST03_541_B69_7.sInit.MaxTime             :=2000;
ST03_541_B69_7.sInit.EnableInEveryMode   :=TRUE;

(* Init ST03_542_B70_0 ISK rechts Lageerkennung (DigIn) *)
ST03_542_B70_0.sInit.InstName            :='ST03_542_B70_0';
ST03_542_B70_0.sInit.Description         :='ISK rechts Lageerkennung';
ST03_542_B70_0.sInit.BitInName           :='+8-542_B70.0';
ST03_542_B70_0.sInit.HomePosSignal       :=2; (* 0: Signal=Low, 1: Signal=High, 2: always  *)
ST03_542_B70_0.sInit.MaxTime             :=2000;
ST03_542_B70_0.sInit.EnableInEveryMode   :=TRUE;

(* Init ST03_542_Y70_1   Zuführung  Vereinzler AST/GST (Valve) *)
ST03_542_Y70_1.sInit.InstName            :='ST03_542_Y70_1';
ST03_542_Y70_1.sInit.BitName            :='+8-542_Y70.1';
ST03_542_Y70_1.sInit.Description         :=' Zuführung Vereinzler AST/GST';
ST03_542_Y70_1.sInit.HomePosDefine       :=HOME_ALWAYS;
ST03_542_Y70_1.sInit.InitDescription     :='GS einfahren';
ST03_542_Y70_1.sInit.WorkDescription     :='AS ausfahren';
ST03_542_Y70_1.sInit.DampBothTime        :=200;
ST03_542_Y70_1.sInit.KindOfValve         :='A';
ST03_542_Y70_1.sInit.MaxTime             :=2000;

(* Init ST03_542_Y70_2   Zuführung  Stopper AST/GST (Valve) *)
ST03_542_Y70_2.sInit.InstName            :='ST03_542_Y70_2';
ST03_542_Y70_2.sInit.BitName            :='+8-542_Y70.2';
ST03_542_Y70_2.sInit.Description         :=' Zuführung Stopper AST/GST';
ST03_542_Y70_2.sInit.HomePosDefine       :=HOME_ALWAYS;
ST03_542_Y70_2.sInit.InitDescription     :='GS ausfahren';
ST03_542_Y70_2.sInit.WorkDescription     :='AS einfahren';
ST03_542_Y70_2.sInit.DampBothTime        :=200;
ST03_542_Y70_2.sInit.KindOfValve         :='A';
ST03_542_Y70_2.sInit.MaxTime             :=2000;
END_ACTION
ACTION Init_206pol:
(*Rüstsatz 206pol*)
(* Init ST03_435_B67_0 Förderbandeinheit  Zuführung Vereinzler AST (ValveSensor) *)
ST03_435_B67_0.sInit.InstName            :='ST03_435_B67_0';
ST03_435_B67_0.sInit.BitName            :='+8_435_B67.0';
ST03_435_B67_0.sInit.Description         :='Förderbandeinheit  Zuführung Vereinzler AST';
ST03_435_B67_0.sInit.SensorType          :=sValveSensorType_INIT;

(* Init ST03_435_B67_1 Förderbandeinheit  Zuführung Vereinzler GST (ValveSensor) *)
ST03_435_B67_1.sInit.InstName            :='ST03_435_B67_1';
ST03_435_B67_1.sInit.BitName            :='+8_435_B67.1';
ST03_435_B67_1.sInit.Description         :='Förderbandeinheit  Zuführung Vereinzler GST';
ST03_435_B67_1.sInit.SensorType          :=sValveSensorType_WORK;

(* Init ST03_435_B67_2 Förderbandeinheit  Zuführung Stopper AST (ValveSensor) *)
ST03_435_B67_2.sInit.InstName            :='ST03_435_B67_2';
ST03_435_B67_2.sInit.BitName            :='+8_435_B67.2';
ST03_435_B67_2.sInit.Description         :='Förderband linke Zuführung Stopper AST';
ST03_435_B67_2.sInit.SensorType          :=sValveSensorType_INIT;

